gfCNCPoint1[21619] = {X 216.8845, Y 71.0993, Z -2.1667, A 0.000, B 0.000, C 0.000 }
gfCNCPoint1[21620] = {X 215.9082, Y 71.0067, Z -2.1667, A 0.000, B 0.000, C 0.000 }
gfCNCPoint1[21621] = {X 214.2382, Y 70.8314, Z -2.1667, A 0.000, B 0.000, C 0.000 }
gfCNCPoint1[21622] = {X 212.6086, Y 70.4263, Z -2.1667, A 0.000, B 0.000, C 0.000 }
gfCNCPoint1[21623] = {X 211.0509, Y 69.7991, Z -2.1667, A 0.000, B 0.000, C 0.000 }
gfCNCPoint1[21624] = {X 209.5953, Y 68.9620, Z -2.1667, A 0.000, B 0.000, C 0.000 }
gfCNCPoint1[21625] = {X 208.2698, Y 67.9311, Z -2.1667, A 0.000, B 0.000, C 0.000 }
gfCNCPoint1[21626] = {X 207.1000, Y 66.7263, Z -2.1667, A 0.000, B 0.000, C 0.000 }
gfCNCPoint1[21627] = {X 206.1086, Y 65.3710, Z -2.1667, A 0.000, B 0.000, C 0.000 }
gfCNCPoint1[21628] = {X 205.3148, Y 63.8913, Z -2.1667, A 0.000, B 0.000, C 0.000 }
gfCNCPoint1[21629] = {X 204.7338, Y 62.3158, Z -2.1667, A 0.000, B 0.000, C 0.000 }
gfCNCPoint1[21630] = {X 204.3769, Y 60.6750, Z -2.1667, A 0.000, B 0.000, C 0.000 }
gfCNCPoint1[21631] = {X 204.2510, Y 59.0005, Z -2.1667, A 0.000, B 0.000, C 0.000 }
gfCNCPoint1[21632] = {X 204.2508, Y 58.0000, Z -2.1667, A 0.000, B 0.000, C 0.000 }
gfCNCPoint1[21633] = {X 204.3397, Y 56.5375, Z -2.1667, A 0.000, B 0.000, C 0.000 }
gfCNCPoint1[21634] = {X 204.6050, Y 55.0964, Z -2.1667, A 0.000, B 0.000, C 0.000 }
gfCNCPoint1[21635] = {X 205.0427, Y 53.6981, Z -2.1667, A 0.000, B 0.000, C 0.000 }
gfCNCPoint1[21636] = {X 205.6466, Y 52.3631, Z -2.1667, A 0.000, B 0.000, C 0.000 }
gfCNCPoint1[21637] = {X 206.5301, Y 50.9380, Z -2.1667, A 0.000, B 0.000, C 0.000 }
gfCNCPoint1[21638] = {X 207.6024, Y 49.6489, Z -2.1667, A 0.000, B 0.000, C 0.000 }
gfCNCPoint1[21639] = {X 208.8429, Y 48.5207, Z -2.1667, A 0.000, B 0.000, C 0.000 }
gfCNCPoint1[21640] = {X 210.2277, Y 47.5751, Z -2.1667, A 0.000, B 0.000, C 0.000 }
gfCNCPoint1[21641] = {X 209.8801, Y 46.3328, Z -2.1667, A 0.000, B 0.000, C 0.000 }
gfCNCPoint1[21642] = {X 209.7572, Y 45.0487, Z -2.1667, A 0.000, B 0.000, C 0.000 }
gfCNCPoint1[21643] = {X 209.7570, Y 44.1994, Z -2.1667, A 0.000, B 0.000, C 0.000 }
gfCNCPoint1[21644] = {X 209.8559, Y 43.0087, Z -2.1667, A 0.000, B 0.000, C 0.000 }
gfCNCPoint1[21645] = {X 210.1499, Y 41.8506, Z -2.1667, A 0.000, B 0.000, C 0.000 }
gfCNCPoint1[21646] = {X 210.6310, Y 40.7569, Z -2.1667, A 0.000, B 0.000, C 0.000 }
gfCNCPoint1[21647] = {X 211.2859, Y 39.7575, Z -2.1667, A 0.000, B 0.000, C 0.000 }
gfCNCPoint1[21648] = {X 211.2859, Y 37.0789, Z -2.1667, A 0.000, B 0.000, C 0.000 }
gfCNCPoint1[21649] = {X 211.2856, Y 17.4412, Z -2.1667, A 0.000, B 0.000, C 0.000 }
gfCNCPoint1[21650] = {X 210.6368, Y 16.4472, Z -2.1667, A 0.000, B 0.000, C 0.000 }
gfCNCPoint1[21651] = {X 210.1581, Y 15.3610, Z -2.1667, A 0.000, B 0.000, C 0.000 }
gfCNCPoint1[21652] = {X 209.8623, Y 14.2115, Z -2.1667, A 0.000, B 0.000, C 0.000 }
gfCNCPoint1[21653] = {X 209.7572, Y 13.0291, Z -2.1667, A 0.000, B 0.000, C 0.000 }
gfCNCPoint1[21654] = {X 209.7570, Y 12.1868, Z -2.1667, A 0.000, B 0.000, C 0.000 }
gfCNCPoint1[21655] = {X 209.7578, Y 12.0809, Z -2.1667, A 0.000, B 0.000, C 0.000 }
gfCNCPoint1[21656] = {X 209.7601, Y 11.9749, Z -2.1667, A 0.000, B 0.000, C 0.000 }
gfCNCPoint1[21657] = {X 209.9068, Y 10.7178, Z -2.1667, A 0.000, B 0.000, C 0.000 }
gfCNCPoint1[21658] = {X 210.2690, Y 9.5051, Z -2.1667, A 0.000, B 0.000, C 0.000 }
gfCNCPoint1[21659] = {X 207.3611, Y 9.5051, Z -2.1667, A 0.000, B 0.000, C 0.000 }
gfCNCPoint1[21660] = {X 207.3611, Y 7.1051, Z -2.1667, A 0.000, B 0.000, C 0.000 }
gfCNCPoint1[21661] = {X 191.1434, Y 7.1051, Z -2.1667, A 0.000, B 0.000, C 0.000 }
gfCNCPoint1[21662] = {X 193.1003, Y 7.6485, Z -2.1667, A 0.000, B 0.000, C 0.000 }
gfCNCPoint1[21663] = {X 194.9835, Y 8.4087, Z -2.1667, A 0.000, B 0.000, C 0.000 }
gfCNCPoint1[21664] = {X 196.7692, Y 9.3759, Z -2.1667, A 0.000, B 0.000, C 0.000 }
gfCNCPoint1[21665] = {X 198.4348, Y 10.5380, Z -2.1667, A 0.000, B 0.000, C 0.000 }
gfCNCPoint1[21666] = {X 198.8568, Y 10.8884, Z -2.1667, A 0.000, B 0.000, C 0.000 }
gfCNCPoint1[21667] = {X 199.2644, Y 11.2556, Z -2.1667, A 0.000, B 0.000, C 0.000 }
gfCNCPoint1[21668] = {X 200.3494, Y 12.3982, Z -2.1667, A 0.000, B 0.000, C 0.000 }
gfCNCPoint1[21669] = {X 201.2950, Y 13.6586, Z -2.1667, A 0.000, B 0.000, C 0.000 }
gfCNCPoint1[21670] = {X 202.0885, Y 15.0198, Z -2.1667, A 0.000, B 0.000, C 0.000 }
gfCNCPoint1[21671] = {X 202.7195, Y 16.4636, Z -2.1667, A 0.000, B 0.000, C 0.000 }
gfCNCPoint1[21672] = {X 203.2132, Y 18.1834, Z -2.1667, A 0.000, B 0.000, C 0.000 }
gfCNCPoint1[21673] = {X 203.5066, Y 19.9484, Z -2.1667, A 0.000, B 0.000, C 0.000 }
gfCNCPoint1[21674] = {X 203.5957, Y 21.7354, Z -2.1667, A 0.000, B 0.000, C 0.000 }
gfCNCPoint1[21675] = {X 203.4793, Y 23.5208, Z -2.1667, A 0.000, B 0.000, C 0.000 }
gfCNCPoint1[21676] = {X 203.1591, Y 25.2812, Z -2.1667, A 0.000, B 0.000, C 0.000 }
gfCNCPoint1[21677] = {X 202.7588, Y 26.6265, Z -2.1667, A 0.000, B 0.000, C 0.000 }
gfCNCPoint1[21678] = {X 202.2073, Y 27.9172, Z -2.1667, A 0.000, B 0.000, C 0.000 }
gfCNCPoint1[21679] = {X 201.5117, Y 29.1363, Z -2.1667, A 0.000, B 0.000, C 0.000 }
gfCNCPoint1[21680] = {X 200.6812, Y 30.2679, Z -2.1667, A 0.000, B 0.000, C 0.000 }
gfCNCPoint1[21681] = {X 199.7268, Y 31.2971, Z -2.1667, A 0.000, B 0.000, C 0.000 }
gfCNCPoint1[21682] = {X 200.5665, Y 31.8696, Z -2.1667, A 0.000, B 0.000, C 0.000 }
gfCNCPoint1[21683] = {X 201.2694, Y 32.6036, Z -2.1667, A 0.000, B 0.000, C 0.000 }
gfCNCPoint1[21684] = {X 201.8050, Y 33.4674, Z -2.1667, A 0.000, B 0.000, C 0.000 }
gfCNCPoint1[21685] = {X 204.8262, Y 39.7091, Z -2.1667, A 0.000, B 0.000, C 0.000 }
gfCNCPoint1[21686] = {X 205.1508, Y 40.5847, Z -2.1667, A 0.000, B 0.000, C 0.000 }
gfCNCPoint1[21687] = {X 205.3026, Y 41.5062, Z -2.1667, A 0.000, B 0.000, C 0.000 }
gfCNCPoint1[21688] = {X 205.2761, Y 42.4397, Z -2.1667, A 0.000, B 0.000, C 0.000 }
gfCNCPoint1[21689] = {X 205.0723, Y 43.3511, Z -2.1667, A 0.000, B 0.000, C 0.000 }
gfCNCPoint1[21690] = {X 204.6986, Y 44.2070, Z -2.1667, A 0.000, B 0.000, C 0.000 }
gfCNCPoint1[21691] = {X 204.1687, Y 44.9760, Z -2.1667, A 0.000, B 0.000, C 0.000 }
gfCNCPoint1[21692] = {X 203.5020, Y 45.6299, Z -2.1667, A 0.000, B 0.000, C 0.000 }
gfCNCPoint1[21693] = {X 202.9655, Y 46.0637, Z -2.1667, A 0.000, B 0.000, C 0.000 }
gfCNCPoint1[21694] = {X 202.2134, Y 46.5637, Z -2.1667, A 0.000, B 0.000, C 0.000 }
gfCNCPoint1[21695] = {X 201.3821, Y 46.9170, Z -2.1667, A 0.000, B 0.000, C 0.000 }
gfCNCPoint1[21696] = {X 200.5002, Y 47.1116, Z -2.1667, A 0.000, B 0.000, C 0.000 }
gfCNCPoint1[21697] = {X 199.5975, Y 47.1409, Z -2.1667, A 0.000, B 0.000, C 0.000 }
gfCNCPoint1[21698] = {X 198.7048, Y 47.0038, Z -2.1667, A 0.000, B 0.000, C 0.000 }
gfCNCPoint1[21699] = {X 196.3906, Y 48.1788, Z -2.1667, A 0.000, B 0.000, C 0.000 }
gfCNCPoint1[21700] = {X 193.9812, Y 49.1436, Z -2.1667, A 0.000, B 0.000, C 0.000 }
gfCNCPoint1[21701] = {X 191.4956, Y 49.8907, Z -2.1667, A 0.000, B 0.000, C 0.000 }
gfCNCPoint1[21702] = {X 190.2923, Y 50.1563, Z -2.1667, A 0.000, B 0.000, C 0.000 }
gfCNCPoint1[21703] = {X 189.0766, Y 50.3577, Z -2.1667, A 0.000, B 0.000, C 0.000 }
gfCNCPoint1[21704] = {X 186.8979, Y 50.5552, Z -2.1667, A 0.000, B 0.000, C 0.000 }
gfCNCPoint1[21705] = {X 184.7103, Y 50.5468, Z -2.1667, A 0.000, B 0.000, C 0.000 }
gfCNCPoint1[21706] = {X 184.7348, Y 50.0675, Z -2.1667, A 0.000, B 0.000, C 0.000 }
gfCNCPoint1[21707] = {X 183.1149, Y 49.9266, Z -2.1667, A 0.000, B 0.000, C 0.000 }
gfCNCPoint1[21708] = {X 181.5093, Y 49.6703, Z -2.1667, A 0.000, B 0.000, C 0.000 }
gfCNCPoint1[21709] = {X 179.6142, Y 49.1965, Z -2.1667, A 0.000, B 0.000, C 0.000 }
gfCNCPoint1[21710] = {X 177.7853, Y 48.5099, Z -2.1667, A 0.000, B 0.000, C 0.000 }
gfCNCPoint1[21711] = {X 176.0466, Y 47.6193, Z -2.1667, A 0.000, B 0.000, C 0.000 }
gfCNCPoint1[21712] = {X 174.4208, Y 46.5365, Z -2.1667, A 0.000, B 0.000, C 0.000 }
gfCNCPoint1[21713] = {X 173.1808, Y 45.4898, Z -2.1667, A 0.000, B 0.000, C 0.000 }
gfCNCPoint1[21714] = {X 172.0773, Y 44.3002, Z -2.1667, A 0.000, B 0.000, C 0.000 }
gfCNCPoint1[21715] = {X 171.1268, Y 42.9851, Z -2.1667, A 0.000, B 0.000, C 0.000 }
gfCNCPoint1[21716] = {X 170.3432, Y 41.5641, Z -2.1667, A 0.000, B 0.000, C 0.000 }
gfCNCPoint1[21717] = {X 169.7384, Y 40.0584, Z -2.1667, A 0.000, B 0.000, C 0.000 }
gfCNCPoint1[21718] = {X 169.3212, Y 38.4903, Z -2.1667, A 0.000, B 0.000, C 0.000 }
gfCNCPoint1[21719] = {X 169.0979, Y 36.8831, Z -2.1667, A 0.000, B 0.000, C 0.000 }
gfCNCPoint1[21720] = {X 169.0134, Y 35.0395, Z -2.1667, A 0.000, B 0.000, C 0.000 }
gfCNCPoint1[21721] = {X 169.1603, Y 33.2000, Z -2.1667, A 0.000, B 0.000, C 0.000 }
gfCNCPoint1[21722] = {X 169.5364, Y 31.3932, Z -2.1667, A 0.000, B 0.000, C 0.000 }
gfCNCPoint1[21723] = {X 170.1356, Y 29.6478, Z -2.1667, A 0.000, B 0.000, C 0.000 }
gfCNCPoint1[21724] = {X 170.7629, Y 28.3601, Z -2.1667, A 0.000, B 0.000, C 0.000 }
gfCNCPoint1[21725] = {X 171.5529, Y 27.1653, Z -2.1667, A 0.000, B 0.000, C 0.000 }
gfCNCPoint1[21726] = {X 172.4921, Y 26.0840, Z -2.1667, A 0.000, B 0.000, C 0.000 }
gfCNCPoint1[21727] = {X 173.5646, Y 25.1346, Z -2.1667, A 0.000, B 0.000, C 0.000 }
gfCNCPoint1[21728] = {X 174.7519, Y 24.3333, Z -2.1667, A 0.000, B 0.000, C 0.000 }
gfCNCPoint1[21729] = {X 173.9915, Y 23.9230, Z -2.1667, A 0.000, B 0.000, C 0.000 }
gfCNCPoint1[21730] = {X 173.3261, Y 23.3721, Z -2.1667, A 0.000, B 0.000, C 0.000 }
gfCNCPoint1[21731] = {X 172.7811, Y 22.7017, Z -2.1667, A 0.000, B 0.000, C 0.000 }
gfCNCPoint1[21732] = {X 172.3776, Y 21.9378, Z -2.1667, A 0.000, B 0.000, C 0.000 }
gfCNCPoint1[21733] = {X 169.7664, Y 15.5423, Z -2.1667, A 0.000, B 0.000, C 0.000 }
gfCNCPoint1[21734] = {X 169.5126, Y 14.6752, Z -2.1667, A 0.000, B 0.000, C 0.000 }
gfCNCPoint1[21735] = {X 169.4412, Y 13.7745, Z -2.1667, A 0.000, B 0.000, C 0.000 }
gfCNCPoint1[21736] = {X 169.5553, Y 12.8782, Z -2.1667, A 0.000, B 0.000, C 0.000 }
gfCNCPoint1[21737] = {X 169.8501, Y 12.0242, Z -2.1667, A 0.000, B 0.000, C 0.000 }
gfCNCPoint1[21738] = {X 170.3131, Y 11.2483, Z -2.1667, A 0.000, B 0.000, C 0.000 }
gfCNCPoint1[21739] = {X 170.9248, Y 10.5834, Z -2.1667, A 0.000, B 0.000, C 0.000 }
gfCNCPoint1[21740] = {X 171.6594, Y 10.0574, Z -2.1667, A 0.000, B 0.000, C 0.000 }
gfCNCPoint1[21741] = {X 172.2916, Y 9.6970, Z -2.1667, A 0.000, B 0.000, C 0.000 }
gfCNCPoint1[21742] = {X 173.1812, Y 9.3215, Z -2.1667, A 0.000, B 0.000, C 0.000 }
gfCNCPoint1[21743] = {X 174.1312, Y 9.1491, Z -2.1667, A 0.000, B 0.000, C 0.000 }
gfCNCPoint1[21744] = {X 175.0960, Y 9.1881, Z -2.1667, A 0.000, B 0.000, C 0.000 }
gfCNCPoint1[21745] = {X 176.0291, Y 9.4366, Z -2.1667, A 0.000, B 0.000, C 0.000 }
gfCNCPoint1[21746] = {X 178.2250, Y 8.5162, Z -2.1667, A 0.000, B 0.000, C 0.000 }
gfCNCPoint1[21747] = {X 180.5019, Y 7.8195, Z -2.1667, A 0.000, B 0.000, C 0.000 }
gfCNCPoint1[21748] = {X 182.8368, Y 7.3533, Z -2.1667, A 0.000, B 0.000, C 0.000 }
gfCNCPoint1[21749] = {X 185.2066, Y 7.1225, Z -2.1667, A 0.000, B 0.000, C 0.000 }
gfCNCPoint1[21750] = {X 187.5877, Y 7.1291, Z -2.1667, A 0.000, B 0.000, C 0.000 }
gfCNCPoint1[21751] = {X 189.9562, Y 7.3732, Z -2.1667, A 0.000, B 0.000, C 0.000 }
gfCNCPoint1[21752] = {X 191.7220, Y 7.7367, Z -2.1667, A 0.000, B 0.000, C 0.000 }
gfCNCPoint1[21753] = {X 193.4411, Y 8.2794, Z -2.1667, A 0.000, B 0.000, C 0.000 }
gfCNCPoint1[21754] = {X 195.0955, Y 8.9958, Z -2.1667, A 0.000, B 0.000, C 0.000 }
gfCNCPoint1[21755] = {X 196.6676, Y 9.8783, Z -2.1667, A 0.000, B 0.000, C 0.000 }
gfCNCPoint1[21756] = {X 198.1408, Y 10.9175, Z -2.1667, A 0.000, B 0.000, C 0.000 }
gfCNCPoint1[21757] = {X 199.2070, Y 11.8672, Z -2.1667, A 0.000, B 0.000, C 0.000 }
gfCNCPoint1[21758] = {X 200.1638, Y 12.9271, Z -2.1667, A 0.000, B 0.000, C 0.000 }
gfCNCPoint1[21759] = {X 200.9999, Y 14.0847, Z -2.1667, A 0.000, B 0.000, C 0.000 }
gfCNCPoint1[21760] = {X 201.7053, Y 15.3261, Z -2.1667, A 0.000, B 0.000, C 0.000 }
gfCNCPoint1[21761] = {X 202.2717, Y 16.6369, Z -2.1667, A 0.000, B 0.000, C 0.000 }
gfCNCPoint1[21762] = {X 202.7479, Y 18.3014, Z -2.1667, A 0.000, B 0.000, C 0.000 }
gfCNCPoint1[21763] = {X 203.0305, Y 20.0095, Z -2.1667, A 0.000, B 0.000, C 0.000 }
gfCNCPoint1[21764] = {X 203.1157, Y 21.7387, Z -2.1667, A 0.000, B 0.000, C 0.000 }
gfCNCPoint1[21765] = {X 203.0025, Y 23.4663, Z -2.1667, A 0.000, B 0.000, C 0.000 }
gfCNCPoint1[21766] = {X 202.6923, Y 25.1696, Z -2.1667, A 0.000, B 0.000, C 0.000 }
gfCNCPoint1[21767] = {X 202.2576, Y 26.5985, Z -2.1667, A 0.000, B 0.000, C 0.000 }
gfCNCPoint1[21768] = {X 201.6456, Y 27.9610, Z -2.1667, A 0.000, B 0.000, C 0.000 }
gfCNCPoint1[21769] = {X 200.8659, Y 29.2349, Z -2.1667, A 0.000, B 0.000, C 0.000 }
gfCNCPoint1[21770] = {X 199.9311, Y 30.3999, Z -2.1667, A 0.000, B 0.000, C 0.000 }
gfCNCPoint1[21771] = {X 198.8564, Y 31.4371, Z -2.1667, A 0.000, B 0.000, C 0.000 }
gfCNCPoint1[21772] = {X 199.6398, Y 31.7988, Z -2.1667, A 0.000, B 0.000, C 0.000 }
gfCNCPoint1[21773] = {X 200.3375, Y 32.3064, Z -2.1667, A 0.000, B 0.000, C 0.000 }
gfCNCPoint1[21774] = {X 200.9227, Y 32.9404, Z -2.1667, A 0.000, B 0.000, C 0.000 }
gfCNCPoint1[21775] = {X 201.3730, Y 33.6764, Z -2.1667, A 0.000, B 0.000, C 0.000 }
gfCNCPoint1[21776] = {X 204.3942, Y 39.9182, Z -2.1667, A 0.000, B 0.000, C 0.000 }
gfCNCPoint1[21777] = {X 204.7207, Y 40.8441, Z -2.1667, A 0.000, B 0.000, C 0.000 }
gfCNCPoint1[21778] = {X 204.8337, Y 41.8194, Z -2.1667, A 0.000, B 0.000, C 0.000 }
gfCNCPoint1[21779] = {X 204.7276, Y 42.7955, Z -2.1667, A 0.000, B 0.000, C 0.000 }
gfCNCPoint1[21780] = {X 204.4078, Y 43.7238, Z -2.1667, A 0.000, B 0.000, C 0.000 }
gfCNCPoint1[21781] = {X 203.8900, Y 44.5580, Z -2.1667, A 0.000, B 0.000, C 0.000 }
gfCNCPoint1[21782] = {X 203.2002, Y 45.2567, Z -2.1667, A 0.000, B 0.000, C 0.000 }
gfCNCPoint1[21783] = {X 202.6637, Y 45.6904, Z -2.1667, A 0.000, B 0.000, C 0.000 }
gfCNCPoint1[21784] = {X 201.9521, Y 46.1590, Z -2.1667, A 0.000, B 0.000, C 0.000 }
gfCNCPoint1[21785] = {X 201.1638, Y 46.4822, Z -2.1667, A 0.000, B 0.000, C 0.000 }
gfCNCPoint1[21786] = {X 200.3280, Y 46.6480, Z -2.1667, A 0.000, B 0.000, C 0.000 }
gfCNCPoint1[21787] = {X 199.4760, Y 46.6501, Z -2.1667, A 0.000, B 0.000, C 0.000 }
gfCNCPoint1[21788] = {X 198.6394, Y 46.4887, Z -2.1667, A 0.000, B 0.000, C 0.000 }
gfCNCPoint1[21789] = {X 196.3113, Y 47.6875, Z -2.1667, A 0.000, B 0.000, C 0.000 }
gfCNCPoint1[21790] = {X 193.8835, Y 48.6692, Z -2.1667, A 0.000, B 0.000, C 0.000 }
gfCNCPoint1[21791] = {X 191.3765, Y 49.4257, Z -2.1667, A 0.000, B 0.000, C 0.000 }
gfCNCPoint1[21792] = {X 189.1872, Y 49.8571, Z -2.1667, A 0.000, B 0.000, C 0.000 }
gfCNCPoint1[21793] = {X 186.9662, Y 50.0717, Z -2.1667, A 0.000, B 0.000, C 0.000 }
gfCNCPoint1[21794] = {X 184.7348, Y 50.0675, Z -2.1667, A 0.000, B 0.000, C 0.000 }
gfCNCPoint1[21795] = {X 184.7103, Y 50.5468, Z -2.1667, A 0.000, B 0.000, C 0.000 }
gfCNCPoint1[21796] = {X 185.7068, Y 51.5003, Z -2.1667, A 0.000, B 0.000, C 0.000 }
gfCNCPoint1[21797] = {X 186.5577, Y 52.5857, Z -2.1667, A 0.000, B 0.000, C 0.000 }
gfCNCPoint1[21798] = {X 187.2457, Y 53.7810, Z -2.1667, A 0.000, B 0.000, C 0.000 }
gfCNCPoint1[21799] = {X 187.7793, Y 55.1333, Z -2.1667, A 0.000, B 0.000, C 0.000 }
gfCNCPoint1[21800] = {X 188.1043, Y 56.5503, Z -2.1667, A 0.000, B 0.000, C 0.000 }
gfCNCPoint1[21801] = {X 188.2135, Y 58.0000, Z -2.1667, A 0.000, B 0.000, C 0.000 }
gfCNCPoint1[21802] = {X 188.2132, Y 59.0140, Z -2.1667, A 0.000, B 0.000, C 0.000 }
gfCNCPoint1[21803] = {X 188.2026, Y 59.3931, Z -2.1667, A 0.000, B 0.000, C 0.000 }
gfCNCPoint1[21804] = {X 188.1772, Y 59.7715, Z -2.1667, A 0.000, B 0.000, C 0.000 }
gfCNCPoint1[21805] = {X 213.5228, Y 87.4328, Z -2.1667, A 0.000, B 0.000, C 0.000 }
gfCNCPoint1[21806] = {X 214.2178, Y 87.3803, Z -2.1667, A 0.000, B 0.000, C 0.000 }
gfCNCPoint1[21807] = {X 214.9136, Y 87.3388, Z -2.1667, A 0.000, B 0.000, C 0.000 }
gfCNCPoint1[21808] = {X 234.0929, Y 75.0516, Z -2.1667, A 0.000, B 0.000, C 0.000 }
gfCNCPoint1[21809] = {X 219.6587, Y 69.3868, Z -2.1667, A 0.000, B 0.000, C 0.000 }
gfCNCPoint1[21810] = {X 218.4698, Y 68.9869, Z -2.1667, A 0.000, B 0.000, C 0.000 }
gfCNCPoint1[21811] = {X 217.2429, Y 68.7262, Z -2.1667, A 0.000, B 0.000, C 0.000 }
gfCNCPoint1[21812] = {X 215.9942, Y 68.6082, Z -2.1667, A 0.000, B 0.000, C 0.000 }
gfCNCPoint1[21813] = {X 214.5238, Y 68.4439, Z -2.1667, A 0.000, B 0.000, C 0.000 }
gfCNCPoint1[21814] = {X 213.0956, Y 68.0575, Z -2.1667, A 0.000, B 0.000, C 0.000 }
gfCNCPoint1[21815] = {X 211.7431, Y 67.4579, Z -2.1667, A 0.000, B 0.000, C 0.000 }
gfCNCPoint1[21816] = {X 210.4977, Y 66.6591, Z -2.1667, A 0.000, B 0.000, C 0.000 }
gfCNCPoint1[21817] = {X 209.3885, Y 65.6800, Z -2.1667, A 0.000, B 0.000, C 0.000 }
gfCNCPoint1[21818] = {X 208.4416, Y 64.5432, Z -2.1667, A 0.000, B 0.000, C 0.000 }
gfCNCPoint1[21819] = {X 207.6789, Y 63.2754, Z -2.1667, A 0.000, B 0.000, C 0.000 }
gfCNCPoint1[21820] = {X 207.1184, Y 61.9061, Z -2.1667, A 0.000, B 0.000, C 0.000 }
gfCNCPoint1[21821] = {X 206.7730, Y 60.4675, Z -2.1667, A 0.000, B 0.000, C 0.000 }
gfCNCPoint1[21822] = {X 206.6510, Y 58.9930, Z -2.1667, A 0.000, B 0.000, C 0.000 }
gfCNCPoint1[21823] = {X 206.6508, Y 58.0000, Z -2.1667, A 0.000, B 0.000, C 0.000 }
gfCNCPoint1[21824] = {X 206.7577, Y 56.5655, Z -2.1667, A 0.000, B 0.000, C 0.000 }
gfCNCPoint1[21825] = {X 207.0759, Y 55.1628, Z -2.1667, A 0.000, B 0.000, C 0.000 }
gfCNCPoint1[21826] = {X 207.5986, Y 53.8226, Z -2.1667, A 0.000, B 0.000, C 0.000 }
gfCNCPoint1[21827] = {X 208.3140, Y 52.5747, Z -2.1667, A 0.000, B 0.000, C 0.000 }
gfCNCPoint1[21828] = {X 209.2065, Y 51.4466, Z -2.1667, A 0.000, B 0.000, C 0.000 }
gfCNCPoint1[21829] = {X 210.2563, Y 50.4632, Z -2.1667, A 0.000, B 0.000, C 0.000 }
gfCNCPoint1[21830] = {X 211.4402, Y 49.6463, Z -2.1667, A 0.000, B 0.000, C 0.000 }
gfCNCPoint1[21831] = {X 212.5893, Y 49.0723, Z -2.1667, A 0.000, B 0.000, C 0.000 }
gfCNCPoint1[21832] = {X 213.8042, Y 48.6556, Z -2.1667, A 0.000, B 0.000, C 0.000 }
gfCNCPoint1[21833] = {X 213.2578, Y 48.0874, Z -2.1667, A 0.000, B 0.000, C 0.000 }
gfCNCPoint1[21834] = {X 212.8100, Y 47.4386, Z -2.1667, A 0.000, B 0.000, C 0.000 }
gfCNCPoint1[21835] = {X 212.4725, Y 46.7262, Z -2.1667, A 0.000, B 0.000, C 0.000 }
gfCNCPoint1[21836] = {X 212.2401, Y 45.8965, Z -2.1667, A 0.000, B 0.000, C 0.000 }
gfCNCPoint1[21837] = {X 212.1572, Y 45.0389, Z -2.1667, A 0.000, B 0.000, C 0.000 }
gfCNCPoint1[21838] = {X 212.1570, Y 44.1994, Z -2.1667, A 0.000, B 0.000, C 0.000 }
gfCNCPoint1[21839] = {X 212.2384, Y 43.3175, Z -2.1667, A 0.000, B 0.000, C 0.000 }
gfCNCPoint1[21840] = {X 212.4799, Y 42.4654, Z -2.1667, A 0.000, B 0.000, C 0.000 }
gfCNCPoint1[21841] = {X 212.8733, Y 41.6720, Z -2.1667, A 0.000, B 0.000, C 0.000 }
gfCNCPoint1[21842] = {X 213.4053, Y 40.9639, Z -2.1667, A 0.000, B 0.000, C 0.000 }
gfCNCPoint1[21843] = {X 213.6831, Y 40.6575, Z -2.1667, A 0.000, B 0.000, C 0.000 }
gfCNCPoint1[21844] = {X 213.6859, Y 40.3041, Z -2.1667, A 0.000, B 0.000, C 0.000 }
gfCNCPoint1[21845] = {X 213.6859, Y 17.4645, Z -2.1667, A 0.000, B 0.000, C 0.000 }
gfCNCPoint1[21846] = {X 213.6805, Y 16.7698, Z -2.1667, A 0.000, B 0.000, C 0.000 }
gfCNCPoint1[21847] = {X 213.6802, Y 16.5201, Z -2.1667, A 0.000, B 0.000, C 0.000 }
gfCNCPoint1[21848] = {X 213.0407, Y 15.7787, Z -2.1667, A 0.000, B 0.000, C 0.000 }
gfCNCPoint1[21849] = {X 212.5621, Y 14.9246, Z -2.1667, A 0.000, B 0.000, C 0.000 }
gfCNCPoint1[21850] = {X 212.2635, Y 13.9921, Z -2.1667, A 0.000, B 0.000, C 0.000 }
gfCNCPoint1[21851] = {X 212.1572, Y 13.0188, Z -2.1667, A 0.000, B 0.000, C 0.000 }
gfCNCPoint1[21852] = {X 212.1570, Y 12.1868, Z -2.1667, A 0.000, B 0.000, C 0.000 }
gfCNCPoint1[21853] = {X 212.2436, Y 11.2718, Z -2.1667, A 0.000, B 0.000, C 0.000 }
gfCNCPoint1[21854] = {X 212.5002, Y 10.3892, Z -2.1667, A 0.000, B 0.000, C 0.000 }
gfCNCPoint1[21855] = {X 212.9449, Y 9.5281, Z -2.1667, A 0.000, B 0.000, C 0.000 }
gfCNCPoint1[21856] = {X 213.5510, Y 8.7718, Z -2.1667, A 0.000, B 0.000, C 0.000 }
gfCNCPoint1[21857] = {X 214.2946, Y 8.1503, Z -2.1667, A 0.000, B 0.000, C 0.000 }
gfCNCPoint1[21858] = {X 215.1463, Y 7.6880, Z -2.1667, A 0.000, B 0.000, C 0.000 }
gfCNCPoint1[21859] = {X 216.0727, Y 7.4030, Z -2.1667, A 0.000, B 0.000, C 0.000 }
gfCNCPoint1[21860] = {X 217.0370, Y 7.3068, Z -2.1667, A 0.000, B 0.000, C 0.000 }
gfCNCPoint1[21861] = {X 223.4805, Y 7.3068, Z -2.1667, A 0.000, B 0.000, C 0.000 }
gfCNCPoint1[21862] = {X 224.4448, Y 7.4030, Z -2.1667, A 0.000, B 0.000, C 0.000 }
gfCNCPoint1[21863] = {X 225.3712, Y 7.6880, Z -2.1667, A 0.000, B 0.000, C 0.000 }
gfCNCPoint1[21864] = {X 226.2229, Y 8.1503, Z -2.1667, A 0.000, B 0.000, C 0.000 }
gfCNCPoint1[21865] = {X 226.9665, Y 8.7718, Z -2.1667, A 0.000, B 0.000, C 0.000 }
gfCNCPoint1[21866] = {X 227.5726, Y 9.5281, Z -2.1667, A 0.000, B 0.000, C 0.000 }
gfCNCPoint1[21867] = {X 228.0173, Y 10.3892, Z -2.1667, A 0.000, B 0.000, C 0.000 }
gfCNCPoint1[21868] = {X 228.2739, Y 11.2718, Z -2.1667, A 0.000, B 0.000, C 0.000 }
gfCNCPoint1[21869] = {X 228.3605, Y 12.1868, Z -2.1667, A 0.000, B 0.000, C 0.000 }
gfCNCPoint1[21870] = {X 228.3603, Y 13.0237, Z -2.1667, A 0.000, B 0.000, C 0.000 }
gfCNCPoint1[21871] = {X 228.2528, Y 13.9974, Z -2.1667, A 0.000, B 0.000, C 0.000 }
gfCNCPoint1[21872] = {X 227.9531, Y 14.9300, Z -2.1667, A 0.000, B 0.000, C 0.000 }
gfCNCPoint1[21873] = {X 227.4732, Y 15.7839, Z -2.1667, A 0.000, B 0.000, C 0.000 }
gfCNCPoint1[21874] = {X 226.8323, Y 16.5248, Z -2.1667, A 0.000, B 0.000, C 0.000 }
gfCNCPoint1[21875] = {X 226.8332, Y 40.6629, Z -2.1667, A 0.000, B 0.000, C 0.000 }
gfCNCPoint1[21876] = {X 227.4738, Y 41.4038, Z -2.1667, A 0.000, B 0.000, C 0.000 }
gfCNCPoint1[21877] = {X 227.9535, Y 42.2577, Z -2.1667, A 0.000, B 0.000, C 0.000 }
gfCNCPoint1[21878] = {X 228.2530, Y 43.1903, Z -2.1667, A 0.000, B 0.000, C 0.000 }
gfCNCPoint1[21879] = {X 228.3603, Y 44.1638, Z -2.1667, A 0.000, B 0.000, C 0.000 }
gfCNCPoint1[21880] = {X 228.3605, Y 45.0000, Z -2.1667, A 0.000, B 0.000, C 0.000 }
gfCNCPoint1[21881] = {X 228.3507, Y 45.3090, Z -2.1667, A 0.000, B 0.000, C 0.000 }
gfCNCPoint1[21882] = {X 228.3214, Y 45.6167, Z -2.1667, A 0.000, B 0.000, C 0.000 }
gfCNCPoint1[21883] = {X 228.0910, Y 46.5992, Z -2.1667, A 0.000, B 0.000, C 0.000 }
gfCNCPoint1[21884] = {X 227.6635, Y 47.5134, Z -2.1667, A 0.000, B 0.000, C 0.000 }
gfCNCPoint1[21885] = {X 227.0571, Y 48.3200, Z -2.1667, A 0.000, B 0.000, C 0.000 }
gfCNCPoint1[21886] = {X 226.7053, Y 47.9934, Z -2.1667, A 0.000, B 0.000, C 0.000 }
gfCNCPoint1[21887] = {X 226.0261, Y 48.5889, Z -2.1667, A 0.000, B 0.000, C 0.000 }
gfCNCPoint1[21888] = {X 225.2396, Y 49.0331, Z -2.1667, A 0.000, B 0.000, C 0.000 }
gfCNCPoint1[21889] = {X 224.3790, Y 49.3073, Z -2.1667, A 0.000, B 0.000, C 0.000 }
gfCNCPoint1[21890] = {X 223.4805, Y 49.4000, Z -2.1667, A 0.000, B 0.000, C 0.000 }
gfCNCPoint1[21891] = {X 217.0370, Y 49.4000, Z -2.1667, A 0.000, B 0.000, C 0.000 }
gfCNCPoint1[21892] = {X 216.0579, Y 49.2897, Z -2.1667, A 0.000, B 0.000, C 0.000 }
gfCNCPoint1[21893] = {X 215.1279, Y 48.9643, Z -2.1667, A 0.000, B 0.000, C 0.000 }
gfCNCPoint1[21894] = {X 214.2936, Y 48.4400, Z -2.1667, A 0.000, B 0.000, C 0.000 }
gfCNCPoint1[21895] = {X 213.5969, Y 47.7433, Z -2.1667, A 0.000, B 0.000, C 0.000 }
gfCNCPoint1[21896] = {X 213.0727, Y 46.9091, Z -2.1667, A 0.000, B 0.000, C 0.000 }
gfCNCPoint1[21897] = {X 212.7473, Y 45.9791, Z -2.1667, A 0.000, B 0.000, C 0.000 }
gfCNCPoint1[21898] = {X 212.6370, Y 45.0000, Z -2.1667, A 0.000, B 0.000, C 0.000 }
gfCNCPoint1[21899] = {X 212.6370, Y 44.1994, Z -2.1667, A 0.000, B 0.000, C 0.000 }
gfCNCPoint1[21900] = {X 212.7103, Y 43.4054, Z -2.1667, A 0.000, B 0.000, C 0.000 }
gfCNCPoint1[21901] = {X 212.9277, Y 42.6382, Z -2.1667, A 0.000, B 0.000, C 0.000 }
gfCNCPoint1[21902] = {X 213.2819, Y 41.9238, Z -2.1667, A 0.000, B 0.000, C 0.000 }
gfCNCPoint1[21903] = {X 213.7609, Y 41.2863, Z -2.1667, A 0.000, B 0.000, C 0.000 }
gfCNCPoint1[21904] = {X 214.1617, Y 40.8442, Z -2.1667, A 0.000, B 0.000, C 0.000 }
gfCNCPoint1[21905] = {X 214.1659, Y 40.3060, Z -2.1667, A 0.000, B 0.000, C 0.000 }
gfCNCPoint1[21906] = {X 214.1659, Y 17.4626, Z -2.1667, A 0.000, B 0.000, C 0.000 }
gfCNCPoint1[21907] = {X 214.1605, Y 16.7692, Z -2.1667, A 0.000, B 0.000, C 0.000 }
gfCNCPoint1[21908] = {X 214.1600, Y 16.3071, Z -2.1667, A 0.000, B 0.000, C 0.000 }
gfCNCPoint1[21909] = {X 213.5172, Y 15.6183, Z -2.1667, A 0.000, B 0.000, C 0.000 }
gfCNCPoint1[21910] = {X 213.0358, Y 14.8084, Z -2.1667, A 0.000, B 0.000, C 0.000 }
gfCNCPoint1[21911] = {X 212.7379, Y 13.9146, Z -2.1667, A 0.000, B 0.000, C 0.000 }
gfCNCPoint1[21912] = {X 212.6370, Y 12.9779, Z -2.1667, A 0.000, B 0.000, C 0.000 }
gfCNCPoint1[21913] = {X 212.6370, Y 12.1868, Z -2.1667, A 0.000, B 0.000, C 0.000 }
gfCNCPoint1[21914] = {X 212.7473, Y 11.2077, Z -2.1667, A 0.000, B 0.000, C 0.000 }
gfCNCPoint1[21915] = {X 213.0728, Y 10.2777, Z -2.1667, A 0.000, B 0.000, C 0.000 }
gfCNCPoint1[21916] = {X 213.5970, Y 9.4435, Z -2.1667, A 0.000, B 0.000, C 0.000 }
gfCNCPoint1[21917] = {X 214.2937, Y 8.7468, Z -2.1667, A 0.000, B 0.000, C 0.000 }
gfCNCPoint1[21918] = {X 215.1279, Y 8.2226, Z -2.1667, A 0.000, B 0.000, C 0.000 }
gfCNCPoint1[21919] = {X 216.0579, Y 7.8971, Z -2.1667, A 0.000, B 0.000, C 0.000 }
gfCNCPoint1[21920] = {X 217.0370, Y 7.7868, Z -2.1667, A 0.000, B 0.000, C 0.000 }
gfCNCPoint1[21921] = {X 223.4805, Y 7.7868, Z -2.1667, A 0.000, B 0.000, C 0.000 }
gfCNCPoint1[21922] = {X 224.4596, Y 7.8971, Z -2.1667, A 0.000, B 0.000, C 0.000 }
gfCNCPoint1[21923] = {X 225.3896, Y 8.2226, Z -2.1667, A 0.000, B 0.000, C 0.000 }
gfCNCPoint1[21924] = {X 226.2238, Y 8.7468, Z -2.1667, A 0.000, B 0.000, C 0.000 }
gfCNCPoint1[21925] = {X 226.9205, Y 9.4435, Z -2.1667, A 0.000, B 0.000, C 0.000 }
gfCNCPoint1[21926] = {X 227.4447, Y 10.2777, Z -2.1667, A 0.000, B 0.000, C 0.000 }
gfCNCPoint1[21927] = {X 227.7702, Y 11.2077, Z -2.1667, A 0.000, B 0.000, C 0.000 }
gfCNCPoint1[21928] = {X 227.8805, Y 12.1868, Z -2.1667, A 0.000, B 0.000, C 0.000 }
gfCNCPoint1[21929] = {X 227.8802, Y 13.0233, Z -2.1667, A 0.000, B 0.000, C 0.000 }
gfCNCPoint1[21930] = {X 227.7719, Y 13.9495, Z -2.1667, A 0.000, B 0.000, C 0.000 }
gfCNCPoint1[21931] = {X 227.4708, Y 14.8321, Z -2.1667, A 0.000, B 0.000, C 0.000 }
gfCNCPoint1[21932] = {X 226.9904, Y 15.6314, Z -2.1667, A 0.000, B 0.000, C 0.000 }
gfCNCPoint1[21933] = {X 226.3523, Y 16.3116, Z -2.1667, A 0.000, B 0.000, C 0.000 }
gfCNCPoint1[21934] = {X 226.3532, Y 40.8760, Z -2.1667, A 0.000, B 0.000, C 0.000 }
gfCNCPoint1[21935] = {X 226.9978, Y 41.5652, Z -2.1667, A 0.000, B 0.000, C 0.000 }
gfCNCPoint1[21936] = {X 227.4805, Y 42.3758, Z -2.1667, A 0.000, B 0.000, C 0.000 }
gfCNCPoint1[21937] = {X 227.7793, Y 43.2708, Z -2.1667, A 0.000, B 0.000, C 0.000 }
gfCNCPoint1[21938] = {X 227.8805, Y 44.2089, Z -2.1667, A 0.000, B 0.000, C 0.000 }
gfCNCPoint1[21939] = {X 227.8805, Y 45.0000, Z -2.1667, A 0.000, B 0.000, C 0.000 }
gfCNCPoint1[21940] = {X 227.8037, Y 45.8182, Z -2.1667, A 0.000, B 0.000, C 0.000 }
gfCNCPoint1[21941] = {X 227.5762, Y 46.6079, Z -2.1667, A 0.000, B 0.000, C 0.000 }
gfCNCPoint1[21942] = {X 227.2057, Y 47.3415, Z -2.1667, A 0.000, B 0.000, C 0.000 }
gfCNCPoint1[21943] = {X 226.7053, Y 47.9934, Z -2.1667, A 0.000, B 0.000, C 0.000 }
gfCNCPoint1[21944] = {X 227.0571, Y 48.3200, Z -2.1667, A 0.000, B 0.000, C 0.000 }
gfCNCPoint1[21945] = {X 236.2309, Y 48.3200, Z -2.1667, A 0.000, B 0.000, C 0.000 }
gfCNCPoint1[21946] = {X 235.6245, Y 47.5134, Z -2.1667, A 0.000, B 0.000, C 0.000 }
gfCNCPoint1[21947] = {X 235.1970, Y 46.5992, Z -2.1667, A 0.000, B 0.000, C 0.000 }
gfCNCPoint1[21948] = {X 234.9666, Y 45.6167, Z -2.1667, A 0.000, B 0.000, C 0.000 }
gfCNCPoint1[21949] = {X 234.9373, Y 45.3090, Z -2.1667, A 0.000, B 0.000, C 0.000 }
gfCNCPoint1[21950] = {X 234.9275, Y 45.0000, Z -2.1667, A 0.000, B 0.000, C 0.000 }
gfCNCPoint1[21951] = {X 234.9275, Y 44.2089, Z -2.1667, A 0.000, B 0.000, C 0.000 }
gfCNCPoint1[21952] = {X 235.0194, Y 43.2661, Z -2.1667, A 0.000, B 0.000, C 0.000 }
gfCNCPoint1[21953] = {X 235.2917, Y 42.3588, Z -2.1667, A 0.000, B 0.000, C 0.000 }
gfCNCPoint1[21954] = {X 235.7342, Y 41.5213, Z -2.1667, A 0.000, B 0.000, C 0.000 }
gfCNCPoint1[21955] = {X 236.3302, Y 40.7849, Z -2.1667, A 0.000, B 0.000, C 0.000 }
gfCNCPoint1[21956] = {X 237.0572, Y 40.1776, Z -2.1667, A 0.000, B 0.000, C 0.000 }
gfCNCPoint1[21957] = {X 237.8878, Y 39.7222, Z -2.1667, A 0.000, B 0.000, C 0.000 }
gfCNCPoint1[21958] = {X 241.5467, Y 32.5603, Z -2.1667, A 0.000, B 0.000, C 0.000 }
gfCNCPoint1[21959] = {X 240.2124, Y 31.5577, Z -2.1667, A 0.000, B 0.000, C 0.000 }
gfCNCPoint1[21960] = {X 239.0318, Y 30.3779, Z -2.1667, A 0.000, B 0.000, C 0.000 }
gfCNCPoint1[21961] = {X 238.0282, Y 29.0444, Z -2.1667, A 0.000, B 0.000, C 0.000 }
gfCNCPoint1[21962] = {X 237.2215, Y 27.5832, Z -2.1667, A 0.000, B 0.000, C 0.000 }
gfCNCPoint1[21963] = {X 236.6275, Y 26.0235, Z -2.1667, A 0.000, B 0.000, C 0.000 }
gfCNCPoint1[21964] = {X 236.1924, Y 24.1499, Z -2.1667, A 0.000, B 0.000, C 0.000 }
gfCNCPoint1[21965] = {X 235.9705, Y 22.2393, Z -2.1667, A 0.000, B 0.000, C 0.000 }
gfCNCPoint1[21966] = {X 235.9646, Y 20.3158, Z -2.1667, A 0.000, B 0.000, C 0.000 }
gfCNCPoint1[21967] = {X 236.1749, Y 18.4039, Z -2.1667, A 0.000, B 0.000, C 0.000 }
gfCNCPoint1[21968] = {X 236.5985, Y 16.5277, Z -2.1667, A 0.000, B 0.000, C 0.000 }
gfCNCPoint1[21969] = {X 237.1178, Y 15.0571, Z -2.1667, A 0.000, B 0.000, C 0.000 }
gfCNCPoint1[21970] = {X 237.8175, Y 13.6633, Z -2.1667, A 0.000, B 0.000, C 0.000 }
gfCNCPoint1[21971] = {X 238.6865, Y 12.3682, Z -2.1667, A 0.000, B 0.000, C 0.000 }
gfCNCPoint1[21972] = {X 239.7111, Y 11.1925, Z -2.1667, A 0.000, B 0.000, C 0.000 }
gfCNCPoint1[21973] = {X 240.8753, Y 10.1545, Z -2.1667, A 0.000, B 0.000, C 0.000 }
gfCNCPoint1[21974] = {X 242.1604, Y 9.2707, Z -2.1667, A 0.000, B 0.000, C 0.000 }
gfCNCPoint1[21975] = {X 243.5464, Y 8.5553, Z -2.1667, A 0.000, B 0.000, C 0.000 }
gfCNCPoint1[21976] = {X 245.0111, Y 8.0194, Z -2.1667, A 0.000, B 0.000, C 0.000 }
gfCNCPoint1[21977] = {X 246.5315, Y 7.6715, Z -2.1667, A 0.000, B 0.000, C 0.000 }
gfCNCPoint1[21978] = {X 248.6761, Y 7.3937, Z -2.1667, A 0.000, B 0.000, C 0.000 }
gfCNCPoint1[21979] = {X 250.8370, Y 7.3116, Z -2.1667, A 0.000, B 0.000, C 0.000 }
gfCNCPoint1[21980] = {X 266.7608, Y 7.3116, Z -2.1667, A 0.000, B 0.000, C 0.000 }
gfCNCPoint1[21981] = {X 267.7190, Y 7.4130, Z -2.1667, A 0.000, B 0.000, C 0.000 }
gfCNCPoint1[21982] = {X 268.6386, Y 7.7006, Z -2.1667, A 0.000, B 0.000, C 0.000 }
gfCNCPoint1[21983] = {X 269.4838, Y 8.1632, Z -2.1667, A 0.000, B 0.000, C 0.000 }
gfCNCPoint1[21984] = {X 270.2217, Y 8.7828, Z -2.1667, A 0.000, B 0.000, C 0.000 }
gfCNCPoint1[21985] = {X 270.8236, Y 9.5353, Z -2.1667, A 0.000, B 0.000, C 0.000 }
gfCNCPoint1[21986] = {X 271.2660, Y 10.3913, Z -2.1667, A 0.000, B 0.000, C 0.000 }
gfCNCPoint1[21987] = {X 271.5232, Y 11.2720, Z -2.1667, A 0.000, B 0.000, C 0.000 }
gfCNCPoint1[21988] = {X 271.6110, Y 12.1853, Z -2.1667, A 0.000, B 0.000, C 0.000 }
gfCNCPoint1[21989] = {X 271.6108, Y 13.0282, Z -2.1667, A 0.000, B 0.000, C 0.000 }
gfCNCPoint1[21990] = {X 271.5123, Y 13.9546, Z -2.1667, A 0.000, B 0.000, C 0.000 }
gfCNCPoint1[21991] = {X 271.2396, Y 14.8453, Z -2.1667, A 0.000, B 0.000, C 0.000 }
gfCNCPoint1[21992] = {X 275.6743, Y 16.6820, Z -2.1667, A 0.000, B 0.000, C 0.000 }
gfCNCPoint1[21993] = {X 275.3123, Y 17.4574, Z -2.1667, A 0.000, B 0.000, C 0.000 }
gfCNCPoint1[21994] = {X 274.8831, Y 18.1978, Z -2.1667, A 0.000, B 0.000, C 0.000 }
gfCNCPoint1[21995] = {X 274.8830, Y 38.9888, Z -2.1667, A 0.000, B 0.000, C 0.000 }
gfCNCPoint1[21996] = {X 275.3139, Y 39.7325, Z -2.1667, A 0.000, B 0.000, C 0.000 }
gfCNCPoint1[21997] = {X 275.6771, Y 40.5115, Z -2.1667, A 0.000, B 0.000, C 0.000 }
gfCNCPoint1[21998] = {X 276.0384, Y 39.7367, Z -2.1667, A 0.000, B 0.000, C 0.000 }
gfCNCPoint1[21999] = {X 276.4662, Y 38.9965, Z -2.1667, A 0.000, B 0.000, C 0.000 }
gfCNCPoint1[22000] = {X 276.4658, Y 18.1982, Z -2.1667, A 0.000, B 0.000, C 0.000 }
gfCNCPoint1[22001] = {X 276.0365, Y 17.4576, Z -2.1667, A 0.000, B 0.000, C 0.000 }
gfCNCPoint1[22002] = {X 275.6743, Y 16.6820, Z -2.1667, A 0.000, B 0.000, C 0.000 }
gfCNCPoint1[22003] = {X 273.4570, Y 15.7637, Z -2.1667, A 0.000, B 0.000, C 0.000 }
gfCNCPoint1[22004] = {X 273.0261, Y 16.6345, Z -2.1667, A 0.000, B 0.000, C 0.000 }
gfCNCPoint1[22005] = {X 272.4831, Y 17.4403, Z -2.1667, A 0.000, B 0.000, C 0.000 }
gfCNCPoint1[22006] = {X 272.4830, Y 39.7463, Z -2.1667, A 0.000, B 0.000, C 0.000 }
gfCNCPoint1[22007] = {X 273.0274, Y 40.5545, Z -2.1667, A 0.000, B 0.000, C 0.000 }
gfCNCPoint1[22008] = {X 273.4591, Y 41.4282, Z -2.1667, A 0.000, B 0.000, C 0.000 }
gfCNCPoint1[22009] = {X 273.7590, Y 42.3100, Z -2.1667, A 0.000, B 0.000, C 0.000 }
gfCNCPoint1[22010] = {X 273.9440, Y 43.2228, Z -2.1667, A 0.000, B 0.000, C 0.000 }
gfCNCPoint1[22011] = {X 274.0108, Y 44.1519, Z -2.1667, A 0.000, B 0.000, C 0.000 }
gfCNCPoint1[22012] = {X 274.0110, Y 45.0000, Z -2.1667, A 0.000, B 0.000, C 0.000 }
gfCNCPoint1[22013] = {X 273.9884, Y 45.5734, Z -2.1667, A 0.000, B 0.000, C 0.000 }
gfCNCPoint1[22014] = {X 273.9207, Y 46.1433, Z -2.1667, A 0.000, B 0.000, C 0.000 }
gfCNCPoint1[22015] = {X 275.0713, Y 45.9760, Z -2.1667, A 0.000, B 0.000, C 0.000 }
gfCNCPoint1[22016] = {X 276.2327, Y 45.9200, Z -2.1667, A 0.000, B 0.000, C 0.000 }
gfCNCPoint1[22017] = {X 277.3960, Y 45.9200, Z -2.1667, A 0.000, B 0.000, C 0.000 }
gfCNCPoint1[22018] = {X 277.3539, Y 45.4857, Z -2.1667, A 0.000, B 0.000, C 0.000 }
gfCNCPoint1[22019] = {X 277.3378, Y 45.0497, Z -2.1667, A 0.000, B 0.000, C 0.000 }
gfCNCPoint1[22020] = {X 277.3377, Y 44.1969, Z -2.1667, A 0.000, B 0.000, C 0.000 }
gfCNCPoint1[22021] = {X 277.4034, Y 43.2528, Z -2.1667, A 0.000, B 0.000, C 0.000 }
gfCNCPoint1[22022] = {X 277.5901, Y 42.3251, Z -2.1667, A 0.000, B 0.000, C 0.000 }
gfCNCPoint1[22023] = {X 277.8948, Y 41.4291, Z -2.1667, A 0.000, B 0.000, C 0.000 }
gfCNCPoint1[22024] = {X 278.3248, Y 40.5581, Z -2.1667, A 0.000, B 0.000, C 0.000 }
gfCNCPoint1[22025] = {X 278.8662, Y 39.7516, Z -2.1667, A 0.000, B 0.000, C 0.000 }
gfCNCPoint1[22026] = {X 278.8658, Y 17.4406, Z -2.1667, A 0.000, B 0.000, C 0.000 }
gfCNCPoint1[22027] = {X 278.3227, Y 16.6347, Z -2.1667, A 0.000, B 0.000, C 0.000 }
gfCNCPoint1[22028] = {X 277.8917, Y 15.7637, Z -2.1667, A 0.000, B 0.000, C 0.000 }
gfCNCPoint1[22029] = {X 277.5902, Y 14.8788, Z -2.1667, A 0.000, B 0.000, C 0.000 }
gfCNCPoint1[22030] = {X 277.4046, Y 13.9627, Z -2.1667, A 0.000, B 0.000, C 0.000 }
gfCNCPoint1[22031] = {X 277.3379, Y 13.0303, Z -2.1667, A 0.000, B 0.000, C 0.000 }
gfCNCPoint1[22032] = {X 277.3377, Y 12.1868, Z -2.1667, A 0.000, B 0.000, C 0.000 }
gfCNCPoint1[22033] = {X 277.3952, Y 11.2737, Z -2.1667, A 0.000, B 0.000, C 0.000 }
gfCNCPoint1[22034] = {X 277.5667, Y 10.3751, Z -2.1667, A 0.000, B 0.000, C 0.000 }
gfCNCPoint1[22035] = {X 277.8496, Y 9.5051, Z -2.1667, A 0.000, B 0.000, C 0.000 }
gfCNCPoint1[22036] = {X 273.4964, Y 9.5051, Z -2.1667, A 0.000, B 0.000, C 0.000 }
gfCNCPoint1[22037] = {X 273.7797, Y 10.3731, Z -2.1667, A 0.000, B 0.000, C 0.000 }
gfCNCPoint1[22038] = {X 273.9521, Y 11.2698, Z -2.1667, A 0.000, B 0.000, C 0.000 }
gfCNCPoint1[22039] = {X 274.0110, Y 12.1809, Z -2.1667, A 0.000, B 0.000, C 0.000 }
gfCNCPoint1[22040] = {X 274.0106, Y 13.0529, Z -2.1667, A 0.000, B 0.000, C 0.000 }
gfCNCPoint1[22041] = {X 273.9421, Y 13.9776, Z -2.1667, A 0.000, B 0.000, C 0.000 }
gfCNCPoint1[22042] = {X 273.7565, Y 14.8861, Z -2.1667, A 0.000, B 0.000, C 0.000 }
gfCNCPoint1[22043] = {X 273.4570, Y 15.7637, Z -2.1667, A 0.000, B 0.000, C 0.000 }
gfCNCPoint1[22044] = {X 271.2396, Y 14.8453, Z -2.1667, A 0.000, B 0.000, C 0.000 }
gfCNCPoint1[22045] = {X 270.7501, Y 15.7460, Z -2.1667, A 0.000, B 0.000, C 0.000 }
gfCNCPoint1[22046] = {X 270.0831, Y 16.5245, Z -2.1667, A 0.000, B 0.000, C 0.000 }
gfCNCPoint1[22047] = {X 270.0829, Y 40.6621, Z -2.1667, A 0.000, B 0.000, C 0.000 }
gfCNCPoint1[22048] = {X 270.7238, Y 41.4030, Z -2.1667, A 0.000, B 0.000, C 0.000 }
gfCNCPoint1[22049] = {X 271.2037, Y 42.2570, Z -2.1667, A 0.000, B 0.000, C 0.000 }
gfCNCPoint1[22050] = {X 271.5034, Y 43.1896, Z -2.1667, A 0.000, B 0.000, C 0.000 }
gfCNCPoint1[22051] = {X 271.6108, Y 44.1633, Z -2.1667, A 0.000, B 0.000, C 0.000 }
gfCNCPoint1[22052] = {X 271.6110, Y 45.0000, Z -2.1667, A 0.000, B 0.000, C 0.000 }
gfCNCPoint1[22053] = {X 271.5959, Y 45.3844, Z -2.1667, A 0.000, B 0.000, C 0.000 }
gfCNCPoint1[22054] = {X 271.5505, Y 45.7664, Z -2.1667, A 0.000, B 0.000, C 0.000 }
gfCNCPoint1[22055] = {X 271.2989, Y 46.7171, Z -2.1667, A 0.000, B 0.000, C 0.000 }
gfCNCPoint1[22056] = {X 270.8619, Y 47.5982, Z -2.1667, A 0.000, B 0.000, C 0.000 }
gfCNCPoint1[22057] = {X 270.2571, Y 48.3736, Z -2.1667, A 0.000, B 0.000, C 0.000 }
gfCNCPoint1[22058] = {X 269.5090, Y 49.0121, Z -2.1667, A 0.000, B 0.000, C 0.000 }
gfCNCPoint1[22059] = {X 268.6482, Y 49.4876, Z -2.1667, A 0.000, B 0.000, C 0.000 }
gfCNCPoint1[22060] = {X 267.7095, Y 49.7809, Z -2.1667, A 0.000, B 0.000, C 0.000 }
gfCNCPoint1[22061] = {X 266.7310, Y 49.8800, Z -2.1667, A 0.000, B 0.000, C 0.000 }
gfCNCPoint1[22062] = {X 262.1384, Y 49.8800, Z -2.1667, A 0.000, B 0.000, C 0.000 }
gfCNCPoint1[22063] = {X 262.1384, Y 54.6800, Z -2.1667, A 0.000, B 0.000, C 0.000 }
gfCNCPoint1[22064] = {X 260.2788, Y 54.6800, Z -2.1667, A 0.000, B 0.000, C 0.000 }
gfCNCPoint1[22065] = {X 261.9952, Y 55.3610, Z -2.1667, A 0.000, B 0.000, C 0.000 }
gfCNCPoint1[22066] = {X 262.0627, Y 55.0197, Z -2.1667, A 0.000, B 0.000, C 0.000 }
gfCNCPoint1[22067] = {X 262.1384, Y 54.6800, Z -2.1667, A 0.000, B 0.000, C 0.000 }
gfCNCPoint1[22068] = {X 262.1384, Y 52.2800, Z -2.1667, A 0.000, B 0.000, C 0.000 }
gfCNCPoint1[22069] = {X 260.2810, Y 52.2800, Z -2.1667, A 0.000, B 0.000, C 0.000 }
gfCNCPoint1[22070] = {X 259.1879, Y 52.1965, Z -2.1667, A 0.000, B 0.000, C 0.000 }
gfCNCPoint1[22071] = {X 258.1198, Y 51.9498, Z -2.1667, A 0.000, B 0.000, C 0.000 }
gfCNCPoint1[22072] = {X 257.1008, Y 51.5455, Z -2.1667, A 0.000, B 0.000, C 0.000 }
gfCNCPoint1[22073] = {X 256.1541, Y 50.9927, Z -2.1667, A 0.000, B 0.000, C 0.000 }
gfCNCPoint1[22074] = {X 255.3011, Y 50.3041, Z -2.1667, A 0.000, B 0.000, C 0.000 }
gfCNCPoint1[22075] = {X 253.6573, Y 52.0528, Z -2.1667, A 0.000, B 0.000, C 0.000 }
gfCNCPoint1[22076] = {X 253.4971, Y 51.8987, Z -2.1667, A 0.000, B 0.000, C 0.000 }
gfCNCPoint1[22077] = {X 253.3406, Y 51.7410, Z -2.1667, A 0.000, B 0.000, C 0.000 }
gfCNCPoint1[22078] = {X 253.2748, Y 51.8082, Z -2.1667, A 0.000, B 0.000, C 0.000 }
gfCNCPoint1[22079] = {X 253.2084, Y 51.8747, Z -2.1667, A 0.000, B 0.000, C 0.000 }
gfCNCPoint1[22080] = {X 253.6573, Y 52.0528, Z -2.1667, A 0.000, B 0.000, C 0.000 }
gfCNCPoint1[22081] = {X 255.3011, Y 50.3041, Z -2.1667, A 0.000, B 0.000, C 0.000 }
gfCNCPoint1[22082] = {X 255.1807, Y 50.1883, Z -2.1667, A 0.000, B 0.000, C 0.000 }
gfCNCPoint1[22083] = {X 255.0630, Y 50.0697, Z -2.1667, A 0.000, B 0.000, C 0.000 }
gfCNCPoint1[22084] = {X 254.3405, Y 49.1989, Z -2.1667, A 0.000, B 0.000, C 0.000 }
gfCNCPoint1[22085] = {X 253.7617, Y 48.2267, Z -2.1667, A 0.000, B 0.000, C 0.000 }
gfCNCPoint1[22086] = {X 253.3406, Y 47.1766, Z -2.1667, A 0.000, B 0.000, C 0.000 }
gfCNCPoint1[22087] = {X 252.9194, Y 48.2267, Z -2.1667, A 0.000, B 0.000, C 0.000 }
gfCNCPoint1[22088] = {X 252.3406, Y 49.1989, Z -2.1667, A 0.000, B 0.000, C 0.000 }
gfCNCPoint1[22089] = {X 251.6182, Y 50.0697, Z -2.1667, A 0.000, B 0.000, C 0.000 }
gfCNCPoint1[22090] = {X 251.5687, Y 50.1202, Z -2.1667, A 0.000, B 0.000, C 0.000 }
gfCNCPoint1[22091] = {X 251.5187, Y 50.1702, Z -2.1667, A 0.000, B 0.000, C 0.000 }
gfCNCPoint1[22092] = {X 250.7132, Y 50.8600, Z -2.1667, A 0.000, B 0.000, C 0.000 }
gfCNCPoint1[22093] = {X 249.8159, Y 51.4254, Z -2.1667, A 0.000, B 0.000, C 0.000 }
gfCNCPoint1[22094] = {X 248.8460, Y 51.8545, Z -2.1667, A 0.000, B 0.000, C 0.000 }
gfCNCPoint1[22095] = {X 247.8241, Y 52.1381, Z -2.1667, A 0.000, B 0.000, C 0.000 }
gfCNCPoint1[22096] = {X 247.8930, Y 52.2640, Z -2.1667, A 0.000, B 0.000, C 0.000 }
gfCNCPoint1[22097] = {X 247.9604, Y 52.3908, Z -2.1667, A 0.000, B 0.000, C 0.000 }
gfCNCPoint1[22098] = {X 250.3413, Y 53.3191, Z -2.1667, A 0.000, B 0.000, C 0.000 }
gfCNCPoint1[22099] = {X 264.1528, Y 58.7991, Z -2.1667, A 0.000, B 0.000, C 0.000 }
gfCNCPoint1[22100] = {X 264.1527, Y 58.0000, Z -2.1667, A 0.000, B 0.000, C 0.000 }
gfCNCPoint1[22101] = {X 264.2034, Y 56.8946, Z -2.1667, A 0.000, B 0.000, C 0.000 }
gfCNCPoint1[22102] = {X 264.3550, Y 55.7984, Z -2.1667, A 0.000, B 0.000, C 0.000 }
gfCNCPoint1[22103] = {X 264.4113, Y 55.5136, Z -2.1667, A 0.000, B 0.000, C 0.000 }
gfCNCPoint1[22104] = {X 264.4745, Y 55.2303, Z -2.1667, A 0.000, B 0.000, C 0.000 }
gfCNCPoint1[22105] = {X 264.9369, Y 53.7185, Z -2.1667, A 0.000, B 0.000, C 0.000 }
gfCNCPoint1[22106] = {X 265.5928, Y 52.2800, Z -2.1667, A 0.000, B 0.000, C 0.000 }
gfCNCPoint1[22107] = {X 262.1384, Y 52.2800, Z -2.1667, A 0.000, B 0.000, C 0.000 }
gfCNCPoint1[22108] = {X 262.1384, Y 49.8800, Z -2.1667, A 0.000, B 0.000, C 0.000 }
gfCNCPoint1[22109] = {X 260.2876, Y 49.8800, Z -2.1667, A 0.000, B 0.000, C 0.000 }
gfCNCPoint1[22110] = {X 259.2646, Y 49.7716, Z -2.1667, A 0.000, B 0.000, C 0.000 }
gfCNCPoint1[22111] = {X 258.2870, Y 49.4511, Z -2.1667, A 0.000, B 0.000, C 0.000 }
gfCNCPoint1[22112] = {X 257.3984, Y 48.9328, Z -2.1667, A 0.000, B 0.000, C 0.000 }
gfCNCPoint1[22113] = {X 256.6382, Y 48.2398, Z -2.1667, A 0.000, B 0.000, C 0.000 }
gfCNCPoint1[22114] = {X 256.0401, Y 47.4028, Z -2.1667, A 0.000, B 0.000, C 0.000 }
gfCNCPoint1[22115] = {X 255.6308, Y 46.4590, Z -2.1667, A 0.000, B 0.000, C 0.000 }
gfCNCPoint1[22116] = {X 255.4666, Y 45.7568, Z -2.1667, A 0.000, B 0.000, C 0.000 }
gfCNCPoint1[22117] = {X 255.4077, Y 45.0380, Z -2.1667, A 0.000, B 0.000, C 0.000 }
gfCNCPoint1[22118] = {X 255.4080, Y 44.1417, Z -2.1667, A 0.000, B 0.000, C 0.000 }
gfCNCPoint1[22119] = {X 255.5183, Y 43.1751, Z -2.1667, A 0.000, B 0.000, C 0.000 }
gfCNCPoint1[22120] = {X 255.8181, Y 42.2497, Z -2.1667, A 0.000, B 0.000, C 0.000 }
gfCNCPoint1[22121] = {X 256.2955, Y 41.4021, Z -2.1667, A 0.000, B 0.000, C 0.000 }
gfCNCPoint1[22122] = {X 256.9315, Y 40.6660, Z -2.1667, A 0.000, B 0.000, C 0.000 }
gfCNCPoint1[22123] = {X 256.9315, Y 35.0338, Z -2.1667, A 0.000, B 0.000, C 0.000 }
gfCNCPoint1[22124] = {X 255.1088, Y 35.0338, Z -2.1667, A 0.000, B 0.000, C 0.000 }
gfCNCPoint1[22125] = {X 251.0863, Y 42.8701, Z -2.1667, A 0.000, B 0.000, C 0.000 }
gfCNCPoint1[22126] = {X 251.2236, Y 43.5125, Z -2.1667, A 0.000, B 0.000, C 0.000 }
gfCNCPoint1[22127] = {X 251.2734, Y 44.1675, Z -2.1667, A 0.000, B 0.000, C 0.000 }
gfCNCPoint1[22128] = {X 251.2736, Y 45.0000, Z -2.1667, A 0.000, B 0.000, C 0.000 }
gfCNCPoint1[22129] = {X 251.2174, Y 45.7380, Z -2.1667, A 0.000, B 0.000, C 0.000 }
gfCNCPoint1[22130] = {X 251.0503, Y 46.4590, Z -2.1667, A 0.000, B 0.000, C 0.000 }
gfCNCPoint1[22131] = {X 250.6346, Y 47.4142, Z -2.1667, A 0.000, B 0.000, C 0.000 }
gfCNCPoint1[22132] = {X 250.0255, Y 48.2593, Z -2.1667, A 0.000, B 0.000, C 0.000 }
gfCNCPoint1[22133] = {X 249.2510, Y 48.9560, Z -2.1667, A 0.000, B 0.000, C 0.000 }
gfCNCPoint1[22134] = {X 248.3462, Y 49.4723, Z -2.1667, A 0.000, B 0.000, C 0.000 }
gfCNCPoint1[22135] = {X 247.3525, Y 49.7849, Z -2.1667, A 0.000, B 0.000, C 0.000 }
gfCNCPoint1[22136] = {X 246.8754, Y 49.8562, Z -2.1667, A 0.000, B 0.000, C 0.000 }
gfCNCPoint1[22137] = {X 246.3936, Y 49.8800, Z -2.1667, A 0.000, B 0.000, C 0.000 }
gfCNCPoint1[22138] = {X 242.5312, Y 49.8800, Z -2.1667, A 0.000, B 0.000, C 0.000 }
gfCNCPoint1[22139] = {X 242.5312, Y 49.4000, Z -2.1667, A 0.000, B 0.000, C 0.000 }
gfCNCPoint1[22140] = {X 239.8075, Y 49.4000, Z -2.1667, A 0.000, B 0.000, C 0.000 }
gfCNCPoint1[22141] = {X 238.8284, Y 49.2897, Z -2.1667, A 0.000, B 0.000, C 0.000 }
gfCNCPoint1[22142] = {X 237.8984, Y 48.9643, Z -2.1667, A 0.000, B 0.000, C 0.000 }
gfCNCPoint1[22143] = {X 237.0641, Y 48.4401, Z -2.1667, A 0.000, B 0.000, C 0.000 }
gfCNCPoint1[22144] = {X 236.3674, Y 47.7434, Z -2.1667, A 0.000, B 0.000, C 0.000 }
gfCNCPoint1[22145] = {X 235.8432, Y 46.9091, Z -2.1667, A 0.000, B 0.000, C 0.000 }
gfCNCPoint1[22146] = {X 235.5178, Y 45.9791, Z -2.1667, A 0.000, B 0.000, C 0.000 }
gfCNCPoint1[22147] = {X 235.4075, Y 45.0000, Z -2.1667, A 0.000, B 0.000, C 0.000 }
gfCNCPoint1[22148] = {X 235.4079, Y 44.1483, Z -2.1667, A 0.000, B 0.000, C 0.000 }
gfCNCPoint1[22149] = {X 235.5063, Y 43.2816, Z -2.1667, A 0.000, B 0.000, C 0.000 }
gfCNCPoint1[22150] = {X 235.7737, Y 42.4514, Z -2.1667, A 0.000, B 0.000, C 0.000 }
gfCNCPoint1[22151] = {X 236.1996, Y 41.6903, Z -2.1667, A 0.000, B 0.000, C 0.000 }
gfCNCPoint1[22152] = {X 236.7672, Y 41.0281, Z -2.1667, A 0.000, B 0.000, C 0.000 }
gfCNCPoint1[22153] = {X 237.4544, Y 40.4909, Z -2.1667, A 0.000, B 0.000, C 0.000 }
gfCNCPoint1[22154] = {X 238.2339, Y 40.0998, Z -2.1667, A 0.000, B 0.000, C 0.000 }
gfCNCPoint1[22155] = {X 242.1752, Y 32.3853, Z -2.1667, A 0.000, B 0.000, C 0.000 }
gfCNCPoint1[22156] = {X 241.0117, Y 31.5929, Z -2.1667, A 0.000, B 0.000, C 0.000 }
gfCNCPoint1[22157] = {X 239.9549, Y 30.6632, Z -2.1667, A 0.000, B 0.000, C 0.000 }
gfCNCPoint1[22158] = {X 239.0207, Y 29.6103, Z -2.1667, A 0.000, B 0.000, C 0.000 }
gfCNCPoint1[22159] = {X 238.2234, Y 28.4503, Z -2.1667, A 0.000, B 0.000, C 0.000 }
gfCNCPoint1[22160] = {X 237.5752, Y 27.2008, Z -2.1667, A 0.000, B 0.000, C 0.000 }
gfCNCPoint1[22161] = {X 237.0859, Y 25.8809, Z -2.1667, A 0.000, B 0.000, C 0.000 }
gfCNCPoint1[22162] = {X 236.6642, Y 24.0613, Z -2.1667, A 0.000, B 0.000, C 0.000 }
gfCNCPoint1[22163] = {X 236.4493, Y 22.2058, Z -2.1667, A 0.000, B 0.000, C 0.000 }
gfCNCPoint1[22164] = {X 236.4441, Y 20.3379, Z -2.1667, A 0.000, B 0.000, C 0.000 }
gfCNCPoint1[22165] = {X 236.6486, Y 18.4812, Z -2.1667, A 0.000, B 0.000, C 0.000 }
gfCNCPoint1[22166] = {X 237.0602, Y 16.6592, Z -2.1667, A 0.000, B 0.000, C 0.000 }
gfCNCPoint1[22167] = {X 237.6343, Y 15.0731, Z -2.1667, A 0.000, B 0.000, C 0.000 }
gfCNCPoint1[22168] = {X 238.4264, Y 13.5838, Z -2.1667, A 0.000, B 0.000, C 0.000 }
gfCNCPoint1[22169] = {X 239.4207, Y 12.2212, Z -2.1667, A 0.000, B 0.000, C 0.000 }
gfCNCPoint1[22170] = {X 240.5974, Y 11.0125, Z -2.1667, A 0.000, B 0.000, C 0.000 }
gfCNCPoint1[22171] = {X 241.9328, Y 9.9819, Z -2.1667, A 0.000, B 0.000, C 0.000 }
gfCNCPoint1[22172] = {X 243.4002, Y 9.1500, Z -2.1667, A 0.000, B 0.000, C 0.000 }
gfCNCPoint1[22173] = {X 244.9704, Y 8.5335, Z -2.1667, A 0.000, B 0.000, C 0.000 }
gfCNCPoint1[22174] = {X 246.6118, Y 8.1447, Z -2.1667, A 0.000, B 0.000, C 0.000 }
gfCNCPoint1[22175] = {X 248.7155, Y 7.8721, Z -2.1667, A 0.000, B 0.000, C 0.000 }
gfCNCPoint1[22176] = {X 250.8352, Y 7.7916, Z -2.1667, A 0.000, B 0.000, C 0.000 }
gfCNCPoint1[22177] = {X 266.7640, Y 7.7916, Z -2.1667, A 0.000, B 0.000, C 0.000 }
gfCNCPoint1[22178] = {X 267.7367, Y 7.9085, Z -2.1667, A 0.000, B 0.000, C 0.000 }
gfCNCPoint1[22179] = {X 268.6595, Y 8.2376, Z -2.1667, A 0.000, B 0.000, C 0.000 }
gfCNCPoint1[22180] = {X 269.4866, Y 8.7626, Z -2.1667, A 0.000, B 0.000, C 0.000 }
gfCNCPoint1[22181] = {X 270.1772, Y 9.4575, Z -2.1667, A 0.000, B 0.000, C 0.000 }
gfCNCPoint1[22182] = {X 270.6970, Y 10.2879, Z -2.1667, A 0.000, B 0.000, C 0.000 }
gfCNCPoint1[22183] = {X 271.0203, Y 11.2127, Z -2.1667, A 0.000, B 0.000, C 0.000 }
gfCNCPoint1[22184] = {X 271.1310, Y 12.1862, Z -2.1667, A 0.000, B 0.000, C 0.000 }
gfCNCPoint1[22185] = {X 271.1308, Y 13.0233, Z -2.1667, A 0.000, B 0.000, C 0.000 }
gfCNCPoint1[22186] = {X 271.0225, Y 13.9495, Z -2.1667, A 0.000, B 0.000, C 0.000 }
gfCNCPoint1[22187] = {X 270.7214, Y 14.8320, Z -2.1667, A 0.000, B 0.000, C 0.000 }
gfCNCPoint1[22188] = {X 270.2411, Y 15.6312, Z -2.1667, A 0.000, B 0.000, C 0.000 }
gfCNCPoint1[22189] = {X 269.6031, Y 16.3113, Z -2.1667, A 0.000, B 0.000, C 0.000 }
gfCNCPoint1[22190] = {X 269.6029, Y 40.8753, Z -2.1667, A 0.000, B 0.000, C 0.000 }
gfCNCPoint1[22191] = {X 270.2478, Y 41.5645, Z -2.1667, A 0.000, B 0.000, C 0.000 }
gfCNCPoint1[22192] = {X 270.7308, Y 42.3753, Z -2.1667, A 0.000, B 0.000, C 0.000 }
gfCNCPoint1[22193] = {X 271.0298, Y 43.2705, Z -2.1667, A 0.000, B 0.000, C 0.000 }
gfCNCPoint1[22194] = {X 271.1310, Y 44.2089, Z -2.1667, A 0.000, B 0.000, C 0.000 }
gfCNCPoint1[22195] = {X 271.1310, Y 45.0000, Z -2.1667, A 0.000, B 0.000, C 0.000 }
gfCNCPoint1[22196] = {X 271.0207, Y 45.9791, Z -2.1667, A 0.000, B 0.000, C 0.000 }
gfCNCPoint1[22197] = {X 270.6953, Y 46.9091, Z -2.1667, A 0.000, B 0.000, C 0.000 }
gfCNCPoint1[22198] = {X 270.1711, Y 47.7434, Z -2.1667, A 0.000, B 0.000, C 0.000 }
gfCNCPoint1[22199] = {X 269.4744, Y 48.4401, Z -2.1667, A 0.000, B 0.000, C 0.000 }
gfCNCPoint1[22200] = {X 268.6401, Y 48.9643, Z -2.1667, A 0.000, B 0.000, C 0.000 }
gfCNCPoint1[22201] = {X 267.7101, Y 49.2897, Z -2.1667, A 0.000, B 0.000, C 0.000 }
gfCNCPoint1[22202] = {X 266.7310, Y 49.4000, Z -2.1667, A 0.000, B 0.000, C 0.000 }
gfCNCPoint1[22203] = {X 260.2876, Y 49.4000, Z -2.1667, A 0.000, B 0.000, C 0.000 }
gfCNCPoint1[22204] = {X 259.3085, Y 49.2897, Z -2.1667, A 0.000, B 0.000, C 0.000 }
gfCNCPoint1[22205] = {X 258.3785, Y 48.9643, Z -2.1667, A 0.000, B 0.000, C 0.000 }
gfCNCPoint1[22206] = {X 257.5442, Y 48.4400, Z -2.1667, A 0.000, B 0.000, C 0.000 }
gfCNCPoint1[22207] = {X 256.8475, Y 47.7433, Z -2.1667, A 0.000, B 0.000, C 0.000 }
gfCNCPoint1[22208] = {X 256.3233, Y 46.9091, Z -2.1667, A 0.000, B 0.000, C 0.000 }
gfCNCPoint1[22209] = {X 255.9979, Y 45.9791, Z -2.1667, A 0.000, B 0.000, C 0.000 }
gfCNCPoint1[22210] = {X 255.8876, Y 45.0000, Z -2.1667, A 0.000, B 0.000, C 0.000 }
gfCNCPoint1[22211] = {X 255.8880, Y 44.1483, Z -2.1667, A 0.000, B 0.000, C 0.000 }
gfCNCPoint1[22212] = {X 255.9984, Y 43.2275, Z -2.1667, A 0.000, B 0.000, C 0.000 }
gfCNCPoint1[22213] = {X 256.2993, Y 42.3503, Z -2.1667, A 0.000, B 0.000, C 0.000 }
gfCNCPoint1[22214] = {X 256.7775, Y 41.5556, Z -2.1667, A 0.000, B 0.000, C 0.000 }
gfCNCPoint1[22215] = {X 257.4115, Y 40.8789, Z -2.1667, A 0.000, B 0.000, C 0.000 }
gfCNCPoint1[22216] = {X 257.4115, Y 34.5538, Z -2.1667, A 0.000, B 0.000, C 0.000 }
gfCNCPoint1[22217] = {X 254.8156, Y 34.5538, Z -2.1667, A 0.000, B 0.000, C 0.000 }
gfCNCPoint1[22218] = {X 250.5701, Y 42.8246, Z -2.1667, A 0.000, B 0.000, C 0.000 }
gfCNCPoint1[22219] = {X 250.7374, Y 43.5078, Z -2.1667, A 0.000, B 0.000, C 0.000 }
gfCNCPoint1[22220] = {X 250.7936, Y 44.2089, Z -2.1667, A 0.000, B 0.000, C 0.000 }
gfCNCPoint1[22221] = {X 250.7936, Y 45.0000, Z -2.1667, A 0.000, B 0.000, C 0.000 }
gfCNCPoint1[22222] = {X 250.6832, Y 45.9791, Z -2.1667, A 0.000, B 0.000, C 0.000 }
gfCNCPoint1[22223] = {X 250.3578, Y 46.9091, Z -2.1667, A 0.000, B 0.000, C 0.000 }
gfCNCPoint1[22224] = {X 249.8336, Y 47.7434, Z -2.1667, A 0.000, B 0.000, C 0.000 }
gfCNCPoint1[22225] = {X 249.1369, Y 48.4401, Z -2.1667, A 0.000, B 0.000, C 0.000 }
gfCNCPoint1[22226] = {X 248.3026, Y 48.9643, Z -2.1667, A 0.000, B 0.000, C 0.000 }
gfCNCPoint1[22227] = {X 247.3727, Y 49.2897, Z -2.1667, A 0.000, B 0.000, C 0.000 }
gfCNCPoint1[22228] = {X 246.3936, Y 49.4000, Z -2.1667, A 0.000, B 0.000, C 0.000 }
gfCNCPoint1[22229] = {X 242.5312, Y 49.4000, Z -2.1667, A 0.000, B 0.000, C 0.000 }
gfCNCPoint1[22230] = {X 242.5312, Y 49.8800, Z -2.1667, A 0.000, B 0.000, C 0.000 }
gfCNCPoint1[22231] = {X 243.4812, Y 50.5824, Z -2.1667, A 0.000, B 0.000, C 0.000 }
gfCNCPoint1[22232] = {X 244.3384, Y 51.3953, Z -2.1667, A 0.000, B 0.000, C 0.000 }
gfCNCPoint1[22233] = {X 245.0903, Y 52.3066, Z -2.1667, A 0.000, B 0.000, C 0.000 }
gfCNCPoint1[22234] = {X 245.7256, Y 53.3027, Z -2.1667, A 0.000, B 0.000, C 0.000 }
gfCNCPoint1[22235] = {X 245.9756, Y 53.7846, Z -2.1667, A 0.000, B 0.000, C 0.000 }
gfCNCPoint1[22236] = {X 246.1982, Y 54.2797, Z -2.1667, A 0.000, B 0.000, C 0.000 }
gfCNCPoint1[22237] = {X 249.4594, Y 55.5512, Z -2.1667, A 0.000, B 0.000, C 0.000 }
gfCNCPoint1[22238] = {X 267.2832, Y 62.6232, Z -2.1667, A 0.000, B 0.000, C 0.000 }
gfCNCPoint1[22239] = {X 266.8848, Y 61.4478, Z -2.1667, A 0.000, B 0.000, C 0.000 }
gfCNCPoint1[22240] = {X 266.6400, Y 60.2311, Z -2.1667, A 0.000, B 0.000, C 0.000 }
gfCNCPoint1[22241] = {X 266.5529, Y 58.9930, Z -2.1667, A 0.000, B 0.000, C 0.000 }
gfCNCPoint1[22242] = {X 266.5527, Y 58.0000, Z -2.1667, A 0.000, B 0.000, C 0.000 }
gfCNCPoint1[22243] = {X 266.6262, Y 56.8093, Z -2.1667, A 0.000, B 0.000, C 0.000 }
gfCNCPoint1[22244] = {X 266.8456, Y 55.6367, Z -2.1667, A 0.000, B 0.000, C 0.000 }
gfCNCPoint1[22245] = {X 267.2076, Y 54.5000, Z -2.1667, A 0.000, B 0.000, C 0.000 }
gfCNCPoint1[22246] = {X 267.7067, Y 53.4164, Z -2.1667, A 0.000, B 0.000, C 0.000 }
gfCNCPoint1[22247] = {X 268.4728, Y 52.2132, Z -2.1667, A 0.000, B 0.000, C 0.000 }
gfCNCPoint1[22248] = {X 269.4075, Y 51.1357, Z -2.1667, A 0.000, B 0.000, C 0.000 }
gfCNCPoint1[22249] = {X 270.4903, Y 50.2072, Z -2.1667, A 0.000, B 0.000, C 0.000 }
gfCNCPoint1[22250] = {X 271.6979, Y 49.4479, Z -2.1667, A 0.000, B 0.000, C 0.000 }
gfCNCPoint1[22251] = {X 273.0039, Y 48.8744, Z -2.1667, A 0.000, B 0.000, C 0.000 }
gfCNCPoint1[22252] = {X 274.3800, Y 48.4989, Z -2.1667, A 0.000, B 0.000, C 0.000 }
gfCNCPoint1[22253] = {X 275.3020, Y 48.3648, Z -2.1667, A 0.000, B 0.000, C 0.000 }
gfCNCPoint1[22254] = {X 276.2327, Y 48.3200, Z -2.1667, A 0.000, B 0.000, C 0.000 }
gfCNCPoint1[22255] = {X 281.0411, Y 48.3200, Z -2.1667, A 0.000, B 0.000, C 0.000 }
gfCNCPoint1[22256] = {X 280.4347, Y 47.5134, Z -2.1667, A 0.000, B 0.000, C 0.000 }
gfCNCPoint1[22257] = {X 280.0072, Y 46.5992, Z -2.1667, A 0.000, B 0.000, C 0.000 }
gfCNCPoint1[22258] = {X 279.7768, Y 45.6167, Z -2.1667, A 0.000, B 0.000, C 0.000 }
gfCNCPoint1[22259] = {X 279.7488, Y 45.3288, Z -2.1667, A 0.000, B 0.000, C 0.000 }
gfCNCPoint1[22260] = {X 279.7378, Y 45.0398, Z -2.1667, A 0.000, B 0.000, C 0.000 }
gfCNCPoint1[22261] = {X 279.7377, Y 44.2037, Z -2.1667, A 0.000, B 0.000, C 0.000 }
gfCNCPoint1[22262] = {X 279.8426, Y 43.2204, Z -2.1667, A 0.000, B 0.000, C 0.000 }
gfCNCPoint1[22263] = {X 280.1416, Y 42.2777, Z -2.1667, A 0.000, B 0.000, C 0.000 }
gfCNCPoint1[22264] = {X 280.6226, Y 41.4137, Z -2.1667, A 0.000, B 0.000, C 0.000 }
gfCNCPoint1[22265] = {X 281.2662, Y 40.6629, Z -2.1667, A 0.000, B 0.000, C 0.000 }
gfCNCPoint1[22266] = {X 281.2658, Y 16.5248, Z -2.1667, A 0.000, B 0.000, C 0.000 }
gfCNCPoint1[22267] = {X 280.6244, Y 15.7831, Z -2.1667, A 0.000, B 0.000, C 0.000 }
gfCNCPoint1[22268] = {X 280.1443, Y 14.9281, Z -2.1667, A 0.000, B 0.000, C 0.000 }
gfCNCPoint1[22269] = {X 279.8447, Y 13.9945, Z -2.1667, A 0.000, B 0.000, C 0.000 }
gfCNCPoint1[22270] = {X 279.7378, Y 13.0198, Z -2.1667, A 0.000, B 0.000, C 0.000 }
gfCNCPoint1[22271] = {X 279.7377, Y 12.1868, Z -2.1667, A 0.000, B 0.000, C 0.000 }
gfCNCPoint1[22272] = {X 279.8242, Y 11.2718, Z -2.1667, A 0.000, B 0.000, C 0.000 }
gfCNCPoint1[22273] = {X 280.0808, Y 10.3892, Z -2.1667, A 0.000, B 0.000, C 0.000 }
gfCNCPoint1[22274] = {X 280.5255, Y 9.5281, Z -2.1667, A 0.000, B 0.000, C 0.000 }
gfCNCPoint1[22275] = {X 281.1316, Y 8.7718, Z -2.1667, A 0.000, B 0.000, C 0.000 }
gfCNCPoint1[22276] = {X 281.8752, Y 8.1503, Z -2.1667, A 0.000, B 0.000, C 0.000 }
gfCNCPoint1[22277] = {X 282.7270, Y 7.6880, Z -2.1667, A 0.000, B 0.000, C 0.000 }
gfCNCPoint1[22278] = {X 283.6533, Y 7.4030, Z -2.1667, A 0.000, B 0.000, C 0.000 }
gfCNCPoint1[22279] = {X 284.6177, Y 7.3068, Z -2.1667, A 0.000, B 0.000, C 0.000 }
gfCNCPoint1[22280] = {X 291.0611, Y 7.3068, Z -2.1667, A 0.000, B 0.000, C 0.000 }
gfCNCPoint1[22281] = {X 292.0255, Y 7.4030, Z -2.1667, A 0.000, B 0.000, C 0.000 }
gfCNCPoint1[22282] = {X 292.9518, Y 7.6880, Z -2.1667, A 0.000, B 0.000, C 0.000 }
gfCNCPoint1[22283] = {X 293.8036, Y 8.1503, Z -2.1667, A 0.000, B 0.000, C 0.000 }
gfCNCPoint1[22284] = {X 294.5472, Y 8.7718, Z -2.1667, A 0.000, B 0.000, C 0.000 }
gfCNCPoint1[22285] = {X 295.1533, Y 9.5281, Z -2.1667, A 0.000, B 0.000, C 0.000 }
gfCNCPoint1[22286] = {X 295.5980, Y 10.3892, Z -2.1667, A 0.000, B 0.000, C 0.000 }
gfCNCPoint1[22287] = {X 295.8044, Y 11.0397, Z -2.1667, A 0.000, B 0.000, C 0.000 }
gfCNCPoint1[22288] = {X 295.9180, Y 11.7127, Z -2.1667, A 0.000, B 0.000, C 0.000 }
gfCNCPoint1[22289] = {X 295.9354, Y 11.9495, Z -2.1667, A 0.000, B 0.000, C 0.000 }
gfCNCPoint1[22290] = {X 295.9411, Y 12.1868, Z -2.1667, A 0.000, B 0.000, C 0.000 }
gfCNCPoint1[22291] = {X 295.9409, Y 13.0237, Z -2.1667, A 0.000, B 0.000, C 0.000 }
gfCNCPoint1[22292] = {X 295.9342, Y 13.2382, Z -2.1667, A 0.000, B 0.000, C 0.000 }
gfCNCPoint1[22293] = {X 295.9180, Y 13.4521, Z -2.1667, A 0.000, B 0.000, C 0.000 }
gfCNCPoint1[22294] = {X 298.3067, Y 13.6853, Z -2.1667, A 0.000, B 0.000, C 0.000 }
gfCNCPoint1[22295] = {X 298.1360, Y 14.6939, Z -2.1667, A 0.000, B 0.000, C 0.000 }
gfCNCPoint1[22296] = {X 297.8256, Y 15.6687, Z -2.1667, A 0.000, B 0.000, C 0.000 }
gfCNCPoint1[22297] = {X 297.3817, Y 16.5904, Z -2.1667, A 0.000, B 0.000, C 0.000 }
gfCNCPoint1[22298] = {X 296.8129, Y 17.4407, Z -2.1667, A 0.000, B 0.000, C 0.000 }
gfCNCPoint1[22299] = {X 296.8133, Y 19.2365, Z -2.1667, A 0.000, B 0.000, C 0.000 }
gfCNCPoint1[22300] = {X 299.8000, Y 19.2365, Z -2.1667, A 0.000, B 0.000, C 0.000 }
gfCNCPoint1[22301] = {X 299.8002, Y 17.4403, Z -2.1667, A 0.000, B 0.000, C 0.000 }
gfCNCPoint1[22302] = {X 299.2315, Y 16.5901, Z -2.1667, A 0.000, B 0.000, C 0.000 }
gfCNCPoint1[22303] = {X 298.7877, Y 15.6685, Z -2.1667, A 0.000, B 0.000, C 0.000 }
gfCNCPoint1[22304] = {X 298.4773, Y 14.6938, Z -2.1667, A 0.000, B 0.000, C 0.000 }
gfCNCPoint1[22305] = {X 298.3067, Y 13.6853, Z -2.1667, A 0.000, B 0.000, C 0.000 }
gfCNCPoint1[22306] = {X 295.9180, Y 13.4521, Z -2.1667, A 0.000, B 0.000, C 0.000 }
gfCNCPoint1[22307] = {X 295.7559, Y 14.3098, Z -2.1667, A 0.000, B 0.000, C 0.000 }
gfCNCPoint1[22308] = {X 295.4436, Y 15.1248, Z -2.1667, A 0.000, B 0.000, C 0.000 }
gfCNCPoint1[22309] = {X 294.9910, Y 15.8712, Z -2.1667, A 0.000, B 0.000, C 0.000 }
gfCNCPoint1[22310] = {X 294.4127, Y 16.5250, Z -2.1667, A 0.000, B 0.000, C 0.000 }
gfCNCPoint1[22311] = {X 294.4139, Y 21.6365, Z -2.1667, A 0.000, B 0.000, C 0.000 }
gfCNCPoint1[22312] = {X 302.1997, Y 21.6365, Z -2.1667, A 0.000, B 0.000, C 0.000 }
gfCNCPoint1[22313] = {X 302.2003, Y 16.5247, Z -2.1667, A 0.000, B 0.000, C 0.000 }
gfCNCPoint1[22314] = {X 301.6222, Y 15.8709, Z -2.1667, A 0.000, B 0.000, C 0.000 }
gfCNCPoint1[22315] = {X 301.1697, Y 15.1246, Z -2.1667, A 0.000, B 0.000, C 0.000 }
gfCNCPoint1[22316] = {X 300.8575, Y 14.3096, Z -2.1667, A 0.000, B 0.000, C 0.000 }
gfCNCPoint1[22317] = {X 300.6953, Y 13.4521, Z -2.1667, A 0.000, B 0.000, C 0.000 }
gfCNCPoint1[22318] = {X 300.6791, Y 13.2371, Z -2.1667, A 0.000, B 0.000, C 0.000 }
gfCNCPoint1[22319] = {X 300.6724, Y 13.0215, Z -2.1667, A 0.000, B 0.000, C 0.000 }
gfCNCPoint1[22320] = {X 300.6723, Y 12.1868, Z -2.1667, A 0.000, B 0.000, C 0.000 }
gfCNCPoint1[22321] = {X 300.6780, Y 11.9495, Z -2.1667, A 0.000, B 0.000, C 0.000 }
gfCNCPoint1[22322] = {X 300.6953, Y 11.7127, Z -2.1667, A 0.000, B 0.000, C 0.000 }
gfCNCPoint1[22323] = {X 300.8090, Y 11.0397, Z -2.1667, A 0.000, B 0.000, C 0.000 }
gfCNCPoint1[22324] = {X 301.0154, Y 10.3892, Z -2.1667, A 0.000, B 0.000, C 0.000 }
gfCNCPoint1[22325] = {X 301.4601, Y 9.5281, Z -2.1667, A 0.000, B 0.000, C 0.000 }
gfCNCPoint1[22326] = {X 302.0662, Y 8.7718, Z -2.1667, A 0.000, B 0.000, C 0.000 }
gfCNCPoint1[22327] = {X 302.8098, Y 8.1503, Z -2.1667, A 0.000, B 0.000, C 0.000 }
gfCNCPoint1[22328] = {X 303.6616, Y 7.6880, Z -2.1667, A 0.000, B 0.000, C 0.000 }
gfCNCPoint1[22329] = {X 304.5879, Y 7.4030, Z -2.1667, A 0.000, B 0.000, C 0.000 }
gfCNCPoint1[22330] = {X 305.5523, Y 7.3068, Z -2.1667, A 0.000, B 0.000, C 0.000 }
gfCNCPoint1[22331] = {X 311.9957, Y 7.3068, Z -2.1667, A 0.000, B 0.000, C 0.000 }
gfCNCPoint1[22332] = {X 312.9478, Y 7.4006, Z -2.1667, A 0.000, B 0.000, C 0.000 }
gfCNCPoint1[22333] = {X 313.8632, Y 7.6783, Z -2.1667, A 0.000, B 0.000, C 0.000 }
gfCNCPoint1[22334] = {X 314.7069, Y 8.1292, Z -2.1667, A 0.000, B 0.000, C 0.000 }
gfCNCPoint1[22335] = {X 315.4464, Y 8.7361, Z -2.1667, A 0.000, B 0.000, C 0.000 }
gfCNCPoint1[22336] = {X 316.0533, Y 9.4756, Z -2.1667, A 0.000, B 0.000, C 0.000 }
gfCNCPoint1[22337] = {X 316.5043, Y 10.3193, Z -2.1667, A 0.000, B 0.000, C 0.000 }
gfCNCPoint1[22338] = {X 316.7820, Y 11.2348, Z -2.1667, A 0.000, B 0.000, C 0.000 }
gfCNCPoint1[22339] = {X 316.8757, Y 12.1868, Z -2.1667, A 0.000, B 0.000, C 0.000 }
gfCNCPoint1[22340] = {X 316.8755, Y 13.0237, Z -2.1667, A 0.000, B 0.000, C 0.000 }
gfCNCPoint1[22341] = {X 316.7681, Y 13.9974, Z -2.1667, A 0.000, B 0.000, C 0.000 }
gfCNCPoint1[22342] = {X 316.4683, Y 14.9300, Z -2.1667, A 0.000, B 0.000, C 0.000 }
gfCNCPoint1[22343] = {X 315.9883, Y 15.7840, Z -2.1667, A 0.000, B 0.000, C 0.000 }
gfCNCPoint1[22344] = {X 315.3474, Y 16.5249, Z -2.1667, A 0.000, B 0.000, C 0.000 }
gfCNCPoint1[22345] = {X 315.3472, Y 40.6617, Z -2.1667, A 0.000, B 0.000, C 0.000 }
gfCNCPoint1[22346] = {X 315.9886, Y 41.4033, Z -2.1667, A 0.000, B 0.000, C 0.000 }
gfCNCPoint1[22347] = {X 316.4689, Y 42.2581, Z -2.1667, A 0.000, B 0.000, C 0.000 }
gfCNCPoint1[22348] = {X 316.7686, Y 43.1917, Z -2.1667, A 0.000, B 0.000, C 0.000 }
gfCNCPoint1[22349] = {X 316.8755, Y 44.1664, Z -2.1667, A 0.000, B 0.000, C 0.000 }
gfCNCPoint1[22350] = {X 316.8757, Y 45.0000, Z -2.1667, A 0.000, B 0.000, C 0.000 }
gfCNCPoint1[22351] = {X 316.8749, Y 45.0899, Z -2.1667, A 0.000, B 0.000, C 0.000 }
gfCNCPoint1[22352] = {X 316.8724, Y 45.1799, Z -2.1667, A 0.000, B 0.000, C 0.000 }
gfCNCPoint1[22353] = {X 316.8594, Y 45.3987, Z -2.1667, A 0.000, B 0.000, C 0.000 }
gfCNCPoint1[22354] = {X 316.8366, Y 45.6167, Z -2.1667, A 0.000, B 0.000, C 0.000 }
gfCNCPoint1[22355] = {X 316.6062, Y 46.5992, Z -2.1667, A 0.000, B 0.000, C 0.000 }
gfCNCPoint1[22356] = {X 316.1787, Y 47.5134, Z -2.1667, A 0.000, B 0.000, C 0.000 }
gfCNCPoint1[22357] = {X 315.5723, Y 48.3200, Z -2.1667, A 0.000, B 0.000, C 0.000 }
gfCNCPoint1[22358] = {X 315.2205, Y 47.9934, Z -2.1667, A 0.000, B 0.000, C 0.000 }
gfCNCPoint1[22359] = {X 314.5413, Y 48.5889, Z -2.1667, A 0.000, B 0.000, C 0.000 }
gfCNCPoint1[22360] = {X 313.7548, Y 49.0331, Z -2.1667, A 0.000, B 0.000, C 0.000 }
gfCNCPoint1[22361] = {X 312.8942, Y 49.3073, Z -2.1667, A 0.000, B 0.000, C 0.000 }
gfCNCPoint1[22362] = {X 311.9957, Y 49.4000, Z -2.1667, A 0.000, B 0.000, C 0.000 }
gfCNCPoint1[22363] = {X 305.5523, Y 49.4000, Z -2.1667, A 0.000, B 0.000, C 0.000 }
gfCNCPoint1[22364] = {X 304.5732, Y 49.2897, Z -2.1667, A 0.000, B 0.000, C 0.000 }
gfCNCPoint1[22365] = {X 303.6432, Y 48.9643, Z -2.1667, A 0.000, B 0.000, C 0.000 }
gfCNCPoint1[22366] = {X 302.8089, Y 48.4400, Z -2.1667, A 0.000, B 0.000, C 0.000 }
gfCNCPoint1[22367] = {X 302.1122, Y 47.7433, Z -2.1667, A 0.000, B 0.000, C 0.000 }
gfCNCPoint1[22368] = {X 301.5880, Y 46.9091, Z -2.1667, A 0.000, B 0.000, C 0.000 }
gfCNCPoint1[22369] = {X 301.2626, Y 45.9791, Z -2.1667, A 0.000, B 0.000, C 0.000 }
gfCNCPoint1[22370] = {X 301.1523, Y 45.0000, Z -2.1667, A 0.000, B 0.000, C 0.000 }
gfCNCPoint1[22371] = {X 301.1524, Y 44.1991, Z -2.1667, A 0.000, B 0.000, C 0.000 }
gfCNCPoint1[22372] = {X 301.2705, Y 43.2557, Z -2.1667, A 0.000, B 0.000, C 0.000 }
gfCNCPoint1[22373] = {X 301.5738, Y 42.3546, Z -2.1667, A 0.000, B 0.000, C 0.000 }
gfCNCPoint1[22374] = {X 302.0502, Y 41.5318, Z -2.1667, A 0.000, B 0.000, C 0.000 }
gfCNCPoint1[22375] = {X 302.6807, Y 40.8202, Z -2.1667, A 0.000, B 0.000, C 0.000 }
gfCNCPoint1[22376] = {X 302.6807, Y 34.1143, Z -2.1667, A 0.000, B 0.000, C 0.000 }
gfCNCPoint1[22377] = {X 293.9337, Y 34.1143, Z -2.1667, A 0.000, B 0.000, C 0.000 }
gfCNCPoint1[22378] = {X 293.9328, Y 40.8664, Z -2.1667, A 0.000, B 0.000, C 0.000 }
gfCNCPoint1[22379] = {X 294.5727, Y 41.5614, Z -2.1667, A 0.000, B 0.000, C 0.000 }
gfCNCPoint1[22380] = {X 295.0536, Y 42.3746, Z -2.1667, A 0.000, B 0.000, C 0.000 }
gfCNCPoint1[22381] = {X 295.3541, Y 43.2703, Z -2.1667, A 0.000, B 0.000, C 0.000 }
gfCNCPoint1[22382] = {X 295.4611, Y 44.2089, Z -2.1667, A 0.000, B 0.000, C 0.000 }
gfCNCPoint1[22383] = {X 295.4611, Y 45.0000, Z -2.1667, A 0.000, B 0.000, C 0.000 }
gfCNCPoint1[22384] = {X 295.3508, Y 45.9791, Z -2.1667, A 0.000, B 0.000, C 0.000 }
gfCNCPoint1[22385] = {X 295.0254, Y 46.9091, Z -2.1667, A 0.000, B 0.000, C 0.000 }
gfCNCPoint1[22386] = {X 294.5012, Y 47.7434, Z -2.1667, A 0.000, B 0.000, C 0.000 }
gfCNCPoint1[22387] = {X 293.8045, Y 48.4401, Z -2.1667, A 0.000, B 0.000, C 0.000 }
gfCNCPoint1[22388] = {X 292.9702, Y 48.9643, Z -2.1667, A 0.000, B 0.000, C 0.000 }
gfCNCPoint1[22389] = {X 292.0402, Y 49.2897, Z -2.1667, A 0.000, B 0.000, C 0.000 }
gfCNCPoint1[22390] = {X 291.0611, Y 49.4000, Z -2.1667, A 0.000, B 0.000, C 0.000 }
gfCNCPoint1[22391] = {X 284.6177, Y 49.4000, Z -2.1667, A 0.000, B 0.000, C 0.000 }
gfCNCPoint1[22392] = {X 283.6386, Y 49.2897, Z -2.1667, A 0.000, B 0.000, C 0.000 }
gfCNCPoint1[22393] = {X 282.7086, Y 48.9643, Z -2.1667, A 0.000, B 0.000, C 0.000 }
gfCNCPoint1[22394] = {X 281.8743, Y 48.4400, Z -2.1667, A 0.000, B 0.000, C 0.000 }
gfCNCPoint1[22395] = {X 281.1776, Y 47.7433, Z -2.1667, A 0.000, B 0.000, C 0.000 }
gfCNCPoint1[22396] = {X 280.6534, Y 46.9091, Z -2.1667, A 0.000, B 0.000, C 0.000 }
gfCNCPoint1[22397] = {X 280.3280, Y 45.9791, Z -2.1667, A 0.000, B 0.000, C 0.000 }
gfCNCPoint1[22398] = {X 280.2177, Y 45.0000, Z -2.1667, A 0.000, B 0.000, C 0.000 }
gfCNCPoint1[22399] = {X 280.2177, Y 44.2065, Z -2.1667, A 0.000, B 0.000, C 0.000 }
gfCNCPoint1[22400] = {X 280.3230, Y 43.2697, Z -2.1667, A 0.000, B 0.000, C 0.000 }
gfCNCPoint1[22401] = {X 280.6232, Y 42.3760, Z -2.1667, A 0.000, B 0.000, C 0.000 }
gfCNCPoint1[22402] = {X 281.1048, Y 41.5656, Z -2.1667, A 0.000, B 0.000, C 0.000 }
gfCNCPoint1[22403] = {X 281.7462, Y 40.8747, Z -2.1667, A 0.000, B 0.000, C 0.000 }
gfCNCPoint1[22404] = {X 281.7458, Y 16.3116, Z -2.1667, A 0.000, B 0.000, C 0.000 }
gfCNCPoint1[22405] = {X 281.1009, Y 15.6224, Z -2.1667, A 0.000, B 0.000, C 0.000 }
gfCNCPoint1[22406] = {X 280.6179, Y 14.8115, Z -2.1667, A 0.000, B 0.000, C 0.000 }
gfCNCPoint1[22407] = {X 280.3189, Y 13.9163, Z -2.1667, A 0.000, B 0.000, C 0.000 }
gfCNCPoint1[22408] = {X 280.2177, Y 12.9779, Z -2.1667, A 0.000, B 0.000, C 0.000 }
gfCNCPoint1[22409] = {X 280.2177, Y 12.1868, Z -2.1667, A 0.000, B 0.000, C 0.000 }
gfCNCPoint1[22410] = {X 280.3280, Y 11.2077, Z -2.1667, A 0.000, B 0.000, C 0.000 }
gfCNCPoint1[22411] = {X 280.6534, Y 10.2777, Z -2.1667, A 0.000, B 0.000, C 0.000 }
gfCNCPoint1[22412] = {X 281.1776, Y 9.4435, Z -2.1667, A 0.000, B 0.000, C 0.000 }
gfCNCPoint1[22413] = {X 281.8743, Y 8.7468, Z -2.1667, A 0.000, B 0.000, C 0.000 }
gfCNCPoint1[22414] = {X 282.7086, Y 8.2226, Z -2.1667, A 0.000, B 0.000, C 0.000 }
gfCNCPoint1[22415] = {X 283.6386, Y 7.8971, Z -2.1667, A 0.000, B 0.000, C 0.000 }
gfCNCPoint1[22416] = {X 284.6177, Y 7.7868, Z -2.1667, A 0.000, B 0.000, C 0.000 }
gfCNCPoint1[22417] = {X 291.0611, Y 7.7868, Z -2.1667, A 0.000, B 0.000, C 0.000 }
gfCNCPoint1[22418] = {X 292.0402, Y 7.8971, Z -2.1667, A 0.000, B 0.000, C 0.000 }
gfCNCPoint1[22419] = {X 292.9702, Y 8.2226, Z -2.1667, A 0.000, B 0.000, C 0.000 }
gfCNCPoint1[22420] = {X 293.8045, Y 8.7468, Z -2.1667, A 0.000, B 0.000, C 0.000 }
gfCNCPoint1[22421] = {X 294.5012, Y 9.4435, Z -2.1667, A 0.000, B 0.000, C 0.000 }
gfCNCPoint1[22422] = {X 295.0254, Y 10.2777, Z -2.1667, A 0.000, B 0.000, C 0.000 }
gfCNCPoint1[22423] = {X 295.3508, Y 11.2077, Z -2.1667, A 0.000, B 0.000, C 0.000 }
gfCNCPoint1[22424] = {X 295.4611, Y 12.1868, Z -2.1667, A 0.000, B 0.000, C 0.000 }
gfCNCPoint1[22425] = {X 295.4609, Y 13.0233, Z -2.1667, A 0.000, B 0.000, C 0.000 }
gfCNCPoint1[22426] = {X 295.3525, Y 13.9496, Z -2.1667, A 0.000, B 0.000, C 0.000 }
gfCNCPoint1[22427] = {X 295.0513, Y 14.8323, Z -2.1667, A 0.000, B 0.000, C 0.000 }
gfCNCPoint1[22428] = {X 294.5708, Y 15.6317, Z -2.1667, A 0.000, B 0.000, C 0.000 }
gfCNCPoint1[22429] = {X 293.9327, Y 16.3118, Z -2.1667, A 0.000, B 0.000, C 0.000 }
gfCNCPoint1[22430] = {X 293.9340, Y 22.1165, Z -2.1667, A 0.000, B 0.000, C 0.000 }
gfCNCPoint1[22431] = {X 302.6797, Y 22.1165, Z -2.1667, A 0.000, B 0.000, C 0.000 }
gfCNCPoint1[22432] = {X 302.6803, Y 16.3115, Z -2.1667, A 0.000, B 0.000, C 0.000 }
gfCNCPoint1[22433] = {X 302.0355, Y 15.6223, Z -2.1667, A 0.000, B 0.000, C 0.000 }
gfCNCPoint1[22434] = {X 301.5524, Y 14.8115, Z -2.1667, A 0.000, B 0.000, C 0.000 }
gfCNCPoint1[22435] = {X 301.2535, Y 13.9163, Z -2.1667, A 0.000, B 0.000, C 0.000 }
gfCNCPoint1[22436] = {X 301.1523, Y 12.9779, Z -2.1667, A 0.000, B 0.000, C 0.000 }
gfCNCPoint1[22437] = {X 301.1523, Y 12.1868, Z -2.1667, A 0.000, B 0.000, C 0.000 }
gfCNCPoint1[22438] = {X 301.2626, Y 11.2077, Z -2.1667, A 0.000, B 0.000, C 0.000 }
gfCNCPoint1[22439] = {X 301.5880, Y 10.2777, Z -2.1667, A 0.000, B 0.000, C 0.000 }
gfCNCPoint1[22440] = {X 302.1122, Y 9.4435, Z -2.1667, A 0.000, B 0.000, C 0.000 }
gfCNCPoint1[22441] = {X 302.8089, Y 8.7468, Z -2.1667, A 0.000, B 0.000, C 0.000 }
gfCNCPoint1[22442] = {X 303.6432, Y 8.2226, Z -2.1667, A 0.000, B 0.000, C 0.000 }
gfCNCPoint1[22443] = {X 304.5732, Y 7.8971, Z -2.1667, A 0.000, B 0.000, C 0.000 }
gfCNCPoint1[22444] = {X 305.5523, Y 7.7868, Z -2.1667, A 0.000, B 0.000, C 0.000 }
gfCNCPoint1[22445] = {X 311.9957, Y 7.7868, Z -2.1667, A 0.000, B 0.000, C 0.000 }
gfCNCPoint1[22446] = {X 312.9748, Y 7.8971, Z -2.1667, A 0.000, B 0.000, C 0.000 }
gfCNCPoint1[22447] = {X 313.9048, Y 8.2226, Z -2.1667, A 0.000, B 0.000, C 0.000 }
gfCNCPoint1[22448] = {X 314.7391, Y 8.7468, Z -2.1667, A 0.000, B 0.000, C 0.000 }
gfCNCPoint1[22449] = {X 315.4358, Y 9.4435, Z -2.1667, A 0.000, B 0.000, C 0.000 }
gfCNCPoint1[22450] = {X 315.9600, Y 10.2777, Z -2.1667, A 0.000, B 0.000, C 0.000 }
gfCNCPoint1[22451] = {X 316.2854, Y 11.2077, Z -2.1667, A 0.000, B 0.000, C 0.000 }
gfCNCPoint1[22452] = {X 316.3957, Y 12.1868, Z -2.1667, A 0.000, B 0.000, C 0.000 }
gfCNCPoint1[22453] = {X 316.3955, Y 13.0233, Z -2.1667, A 0.000, B 0.000, C 0.000 }
gfCNCPoint1[22454] = {X 316.2871, Y 13.9496, Z -2.1667, A 0.000, B 0.000, C 0.000 }
gfCNCPoint1[22455] = {X 315.9860, Y 14.8322, Z -2.1667, A 0.000, B 0.000, C 0.000 }
gfCNCPoint1[22456] = {X 315.5055, Y 15.6315, Z -2.1667, A 0.000, B 0.000, C 0.000 }
gfCNCPoint1[22457] = {X 314.8674, Y 16.3117, Z -2.1667, A 0.000, B 0.000, C 0.000 }
gfCNCPoint1[22458] = {X 314.8672, Y 40.8749, Z -2.1667, A 0.000, B 0.000, C 0.000 }
gfCNCPoint1[22459] = {X 315.5122, Y 41.5641, Z -2.1667, A 0.000, B 0.000, C 0.000 }
gfCNCPoint1[22460] = {X 315.9954, Y 42.3751, Z -2.1667, A 0.000, B 0.000, C 0.000 }
gfCNCPoint1[22461] = {X 316.2945, Y 43.2704, Z -2.1667, A 0.000, B 0.000, C 0.000 }
gfCNCPoint1[22462] = {X 316.3957, Y 44.2089, Z -2.1667, A 0.000, B 0.000, C 0.000 }
gfCNCPoint1[22463] = {X 316.3957, Y 45.0000, Z -2.1667, A 0.000, B 0.000, C 0.000 }
gfCNCPoint1[22464] = {X 316.3190, Y 45.8182, Z -2.1667, A 0.000, B 0.000, C 0.000 }
gfCNCPoint1[22465] = {X 316.0914, Y 46.6079, Z -2.1667, A 0.000, B 0.000, C 0.000 }
gfCNCPoint1[22466] = {X 315.7209, Y 47.3415, Z -2.1667, A 0.000, B 0.000, C 0.000 }
gfCNCPoint1[22467] = {X 315.2205, Y 47.9934, Z -2.1667, A 0.000, B 0.000, C 0.000 }
gfCNCPoint1[22468] = {X 315.5723, Y 48.3200, Z -2.1667, A 0.000, B 0.000, C 0.000 }
gfCNCPoint1[22469] = {X 324.3107, Y 48.3200, Z -2.1667, A 0.000, B 0.000, C 0.000 }
gfCNCPoint1[22470] = {X 325.5555, Y 48.4004, Z -2.1667, A 0.000, B 0.000, C 0.000 }
gfCNCPoint1[22471] = {X 326.7797, Y 48.6402, Z -2.1667, A 0.000, B 0.000, C 0.000 }
gfCNCPoint1[22472] = {X 325.5882, Y 48.0963, Z -2.1667, A 0.000, B 0.000, C 0.000 }
gfCNCPoint1[22473] = {X 324.4810, Y 47.3966, Z -2.1667, A 0.000, B 0.000, C 0.000 }
gfCNCPoint1[22474] = {X 323.4784, Y 46.5538, Z -2.1667, A 0.000, B 0.000, C 0.000 }
gfCNCPoint1[22475] = {X 322.8382, Y 45.9295, Z -2.1667, A 0.000, B 0.000, C 0.000 }
gfCNCPoint1[22476] = {X 322.2180, Y 45.2650, Z -2.1667, A 0.000, B 0.000, C 0.000 }
gfCNCPoint1[22477] = {X 321.6628, Y 44.5452, Z -2.1667, A 0.000, B 0.000, C 0.000 }
gfCNCPoint1[22478] = {X 323.6300, Y 43.1703, Z -2.1667, A 0.000, B 0.000, C 0.000 }
gfCNCPoint1[22479] = {X 323.0063, Y 42.0918, Z -2.1667, A 0.000, B 0.000, C 0.000 }
gfCNCPoint1[22480] = {X 322.5757, Y 40.9227, Z -2.1667, A 0.000, B 0.000, C 0.000 }
gfCNCPoint1[22481] = {X 322.3506, Y 39.6973, Z -2.1667, A 0.000, B 0.000, C 0.000 }
gfCNCPoint1[22482] = {X 322.3379, Y 38.4514, Z -2.1667, A 0.000, B 0.000, C 0.000 }
gfCNCPoint1[22483] = {X 322.5377, Y 37.2217, Z -2.1667, A 0.000, B 0.000, C 0.000 }
gfCNCPoint1[22484] = {X 322.9443, Y 36.0440, Z -2.1667, A 0.000, B 0.000, C 0.000 }
gfCNCPoint1[22485] = {X 323.5458, Y 34.9529, Z -2.1667, A 0.000, B 0.000, C 0.000 }
gfCNCPoint1[22486] = {X 327.7841, Y 28.6157, Z -2.1667, A 0.000, B 0.000, C 0.000 }
gfCNCPoint1[22487] = {X 328.5200, Y 27.6906, Z -2.1667, A 0.000, B 0.000, C 0.000 }
gfCNCPoint1[22488] = {X 329.3960, Y 26.8968, Z -2.1667, A 0.000, B 0.000, C 0.000 }
gfCNCPoint1[22489] = {X 330.3889, Y 26.2552, Z -2.1667, A 0.000, B 0.000, C 0.000 }
gfCNCPoint1[22490] = {X 331.5063, Y 25.7713, Z -2.1667, A 0.000, B 0.000, C 0.000 }
gfCNCPoint1[22491] = {X 332.6887, Y 25.4804, Z -2.1667, A 0.000, B 0.000, C 0.000 }
gfCNCPoint1[22492] = {X 333.9031, Y 25.3907, Z -2.1667, A 0.000, B 0.000, C 0.000 }
gfCNCPoint1[22493] = {X 335.1154, Y 25.5046, Z -2.1667, A 0.000, B 0.000, C 0.000 }
gfCNCPoint1[22494] = {X 336.2918, Y 25.8191, Z -2.1667, A 0.000, B 0.000, C 0.000 }
gfCNCPoint1[22495] = {X 337.3993, Y 26.3252, Z -2.1667, A 0.000, B 0.000, C 0.000 }
gfCNCPoint1[22496] = {X 338.1754, Y 26.8291, Z -2.1667, A 0.000, B 0.000, C 0.000 }
gfCNCPoint1[22497] = {X 338.8813, Y 27.4275, Z -2.1667, A 0.000, B 0.000, C 0.000 }
gfCNCPoint1[22498] = {X 339.4514, Y 27.9767, Z -2.1667, A 0.000, B 0.000, C 0.000 }
gfCNCPoint1[22499] = {X 339.8232, Y 28.3622, Z -2.1667, A 0.000, B 0.000, C 0.000 }
gfCNCPoint1[22500] = {X 340.1656, Y 28.7740, Z -2.1667, A 0.000, B 0.000, C 0.000 }
gfCNCPoint1[22501] = {X 345.8671, Y 24.3770, Z -2.1667, A 0.000, B 0.000, C 0.000 }
gfCNCPoint1[22502] = {X 346.4662, Y 25.2138, Z -2.1667, A 0.000, B 0.000, C 0.000 }
gfCNCPoint1[22503] = {X 347.0044, Y 26.0909, Z -2.1667, A 0.000, B 0.000, C 0.000 }
gfCNCPoint1[22504] = {X 347.1184, Y 24.7348, Z -2.1667, A 0.000, B 0.000, C 0.000 }
gfCNCPoint1[22505] = {X 346.9945, Y 23.3795, Z -2.1667, A 0.000, B 0.000, C 0.000 }
gfCNCPoint1[22506] = {X 346.9504, Y 23.1695, Z -2.1667, A 0.000, B 0.000, C 0.000 }
gfCNCPoint1[22507] = {X 346.8822, Y 22.9661, Z -2.1667, A 0.000, B 0.000, C 0.000 }
gfCNCPoint1[22508] = {X 346.3958, Y 23.6868, Z -2.1667, A 0.000, B 0.000, C 0.000 }
gfCNCPoint1[22509] = {X 345.8671, Y 24.3770, Z -2.1667, A 0.000, B 0.000, C 0.000 }
gfCNCPoint1[22510] = {X 343.9666, Y 25.8427, Z -2.1667, A 0.000, B 0.000, C 0.000 }
gfCNCPoint1[22511] = {X 344.4664, Y 26.5407, Z -2.1667, A 0.000, B 0.000, C 0.000 }
gfCNCPoint1[22512] = {X 344.9154, Y 27.2725, Z -2.1667, A 0.000, B 0.000, C 0.000 }
gfCNCPoint1[22513] = {X 345.4671, Y 28.3758, Z -2.1667, A 0.000, B 0.000, C 0.000 }
gfCNCPoint1[22514] = {X 345.9034, Y 29.5297, Z -2.1667, A 0.000, B 0.000, C 0.000 }
gfCNCPoint1[22515] = {X 346.4600, Y 29.6323, Z -2.1667, A 0.000, B 0.000, C 0.000 }
gfCNCPoint1[22516] = {X 347.0259, Y 29.6231, Z -2.1667, A 0.000, B 0.000, C 0.000 }
gfCNCPoint1[22517] = {X 347.4365, Y 29.5576, Z -2.1667, A 0.000, B 0.000, C 0.000 }
gfCNCPoint1[22518] = {X 347.7959, Y 29.3488, Z -2.1667, A 0.000, B 0.000, C 0.000 }
gfCNCPoint1[22519] = {X 348.4758, Y 28.6282, Z -2.1667, A 0.000, B 0.000, C 0.000 }
gfCNCPoint1[22520] = {X 348.9864, Y 27.7792, Z -2.1667, A 0.000, B 0.000, C 0.000 }
gfCNCPoint1[22521] = {X 349.3042, Y 26.8409, Z -2.1667, A 0.000, B 0.000, C 0.000 }
gfCNCPoint1[22522] = {X 349.3381, Y 26.6709, Z -2.1667, A 0.000, B 0.000, C 0.000 }
gfCNCPoint1[22523] = {X 349.3692, Y 26.5004, Z -2.1667, A 0.000, B 0.000, C 0.000 }
gfCNCPoint1[22524] = {X 349.5028, Y 25.3288, Z -2.1667, A 0.000, B 0.000, C 0.000 }
gfCNCPoint1[22525] = {X 349.5000, Y 24.1496, Z -2.1667, A 0.000, B 0.000, C 0.000 }
gfCNCPoint1[22526] = {X 349.3609, Y 22.9786, Z -2.1667, A 0.000, B 0.000, C 0.000 }
gfCNCPoint1[22527] = {X 349.1890, Y 22.2868, Z -2.1667, A 0.000, B 0.000, C 0.000 }
gfCNCPoint1[22528] = {X 348.9036, Y 21.6335, Z -2.1667, A 0.000, B 0.000, C 0.000 }
gfCNCPoint1[22529] = {X 348.5128, Y 21.0373, Z -2.1667, A 0.000, B 0.000, C 0.000 }
gfCNCPoint1[22530] = {X 348.1202, Y 20.6779, Z -2.1667, A 0.000, B 0.000, C 0.000 }
gfCNCPoint1[22531] = {X 347.6258, Y 20.4807, Z -2.1667, A 0.000, B 0.000, C 0.000 }
gfCNCPoint1[22532] = {X 346.5729, Y 20.3822, Z -2.1667, A 0.000, B 0.000, C 0.000 }
gfCNCPoint1[22533] = {X 345.5201, Y 20.4825, Z -2.1667, A 0.000, B 0.000, C 0.000 }
gfCNCPoint1[22534] = {X 344.7179, Y 21.8934, Z -2.1667, A 0.000, B 0.000, C 0.000 }
gfCNCPoint1[22535] = {X 343.7339, Y 23.1840, Z -2.1667, A 0.000, B 0.000, C 0.000 }
gfCNCPoint1[22536] = {X 342.5857, Y 24.3311, Z -2.1667, A 0.000, B 0.000, C 0.000 }
gfCNCPoint1[22537] = {X 342.7814, Y 24.5197, Z -2.1667, A 0.000, B 0.000, C 0.000 }
gfCNCPoint1[22538] = {X 343.3984, Y 25.1594, Z -2.1667, A 0.000, B 0.000, C 0.000 }
gfCNCPoint1[22539] = {X 343.9666, Y 25.8427, Z -2.1667, A 0.000, B 0.000, C 0.000 }
gfCNCPoint1[22540] = {X 342.0661, Y 27.3083, Z -2.1667, A 0.000, B 0.000, C 0.000 }
gfCNCPoint1[22541] = {X 342.8615, Y 28.5166, Z -2.1667, A 0.000, B 0.000, C 0.000 }
gfCNCPoint1[22542] = {X 343.4678, Y 29.8299, Z -2.1667, A 0.000, B 0.000, C 0.000 }
gfCNCPoint1[22543] = {X 343.8718, Y 31.2189, Z -2.1667, A 0.000, B 0.000, C 0.000 }
gfCNCPoint1[22544] = {X 344.6368, Y 31.6218, Z -2.1667, A 0.000, B 0.000, C 0.000 }
gfCNCPoint1[22545] = {X 345.4576, Y 31.8938, Z -2.1667, A 0.000, B 0.000, C 0.000 }
gfCNCPoint1[22546] = {X 346.3118, Y 32.0276, Z -2.1667, A 0.000, B 0.000, C 0.000 }
gfCNCPoint1[22547] = {X 347.1765, Y 32.0194, Z -2.1667, A 0.000, B 0.000, C 0.000 }
gfCNCPoint1[22548] = {X 347.9605, Y 31.9042, Z -2.1667, A 0.000, B 0.000, C 0.000 }
gfCNCPoint1[22549] = {X 348.6992, Y 31.6173, Z -2.1667, A 0.000, B 0.000, C 0.000 }
gfCNCPoint1[22550] = {X 349.3554, Y 31.1731, Z -2.1667, A 0.000, B 0.000, C 0.000 }
gfCNCPoint1[22551] = {X 350.1553, Y 30.3690, Z -2.1667, A 0.000, B 0.000, C 0.000 }
gfCNCPoint1[22552] = {X 350.8152, Y 29.4467, Z -2.1667, A 0.000, B 0.000, C 0.000 }
gfCNCPoint1[22553] = {X 351.3180, Y 28.4302, Z -2.1667, A 0.000, B 0.000, C 0.000 }
gfCNCPoint1[22554] = {X 351.6505, Y 27.3459, Z -2.1667, A 0.000, B 0.000, C 0.000 }
gfCNCPoint1[22555] = {X 351.8787, Y 25.7633, Z -2.1667, A 0.000, B 0.000, C 0.000 }
gfCNCPoint1[22556] = {X 351.9042, Y 24.1645, Z -2.1667, A 0.000, B 0.000, C 0.000 }
gfCNCPoint1[22557] = {X 351.7268, Y 22.5754, Z -2.1667, A 0.000, B 0.000, C 0.000 }
gfCNCPoint1[22558] = {X 351.4579, Y 21.5045, Z -2.1667, A 0.000, B 0.000, C 0.000 }
gfCNCPoint1[22559] = {X 351.0152, Y 20.4929, Z -2.1667, A 0.000, B 0.000, C 0.000 }
gfCNCPoint1[22560] = {X 350.4110, Y 19.5687, Z -2.1667, A 0.000, B 0.000, C 0.000 }
gfCNCPoint1[22561] = {X 349.7599, Y 18.9039, Z -2.1667, A 0.000, B 0.000, C 0.000 }
gfCNCPoint1[22562] = {X 348.9693, Y 18.4132, Z -2.1667, A 0.000, B 0.000, C 0.000 }
gfCNCPoint1[22563] = {X 348.0846, Y 18.1249, Z -2.1667, A 0.000, B 0.000, C 0.000 }
gfCNCPoint1[22564] = {X 346.9931, Y 17.9929, Z -2.1667, A 0.000, B 0.000, C 0.000 }
gfCNCPoint1[22565] = {X 345.8939, Y 18.0114, Z -2.1667, A 0.000, B 0.000, C 0.000 }
gfCNCPoint1[22566] = {X 344.8075, Y 18.1799, Z -2.1667, A 0.000, B 0.000, C 0.000 }
gfCNCPoint1[22567] = {X 343.7543, Y 18.4953, Z -2.1667, A 0.000, B 0.000, C 0.000 }
gfCNCPoint1[22568] = {X 343.2662, Y 19.6257, Z -2.1667, A 0.000, B 0.000, C 0.000 }
gfCNCPoint1[22569] = {X 342.6386, Y 20.6850, Z -2.1667, A 0.000, B 0.000, C 0.000 }
gfCNCPoint1[22570] = {X 341.8815, Y 21.6560, Z -2.1667, A 0.000, B 0.000, C 0.000 }
gfCNCPoint1[22571] = {X 341.0073, Y 22.5231, Z -2.1667, A 0.000, B 0.000, C 0.000 }
gfCNCPoint1[22572] = {X 340.7217, Y 22.7629, Z -2.1667, A 0.000, B 0.000, C 0.000 }
gfCNCPoint1[22573] = {X 340.4270, Y 22.9916, Z -2.1667, A 0.000, B 0.000, C 0.000 }
gfCNCPoint1[22574] = {X 339.6615, Y 23.5549, Z -2.1667, A 0.000, B 0.000, C 0.000 }
gfCNCPoint1[22575] = {X 339.1299, Y 23.9121, Z -2.1667, A 0.000, B 0.000, C 0.000 }
gfCNCPoint1[22576] = {X 338.5759, Y 24.2333, Z -2.1667, A 0.000, B 0.000, C 0.000 }
gfCNCPoint1[22577] = {X 339.6078, Y 24.9035, Z -2.1667, A 0.000, B 0.000, C 0.000 }
gfCNCPoint1[22578] = {X 340.5464, Y 25.6991, Z -2.1667, A 0.000, B 0.000, C 0.000 }
gfCNCPoint1[22579] = {X 341.1164, Y 26.2482, Z -2.1667, A 0.000, B 0.000, C 0.000 }
gfCNCPoint1[22580] = {X 341.6108, Y 26.7608, Z -2.1667, A 0.000, B 0.000, C 0.000 }
gfCNCPoint1[22581] = {X 342.0661, Y 27.3083, Z -2.1667, A 0.000, B 0.000, C 0.000 }
gfCNCPoint1[22582] = {X 340.1656, Y 28.7740, Z -2.1667, A 0.000, B 0.000, C 0.000 }
gfCNCPoint1[22583] = {X 340.7342, Y 29.6299, Z -2.1667, A 0.000, B 0.000, C 0.000 }
gfCNCPoint1[22584] = {X 341.1765, Y 30.5574, Z -2.1667, A 0.000, B 0.000, C 0.000 }
gfCNCPoint1[22585] = {X 341.4839, Y 31.5378, Z -2.1667, A 0.000, B 0.000, C 0.000 }
gfCNCPoint1[22586] = {X 341.6501, Y 32.5518, Z -2.1667, A 0.000, B 0.000, C 0.000 }
gfCNCPoint1[22587] = {X 341.8441, Y 32.7094, Z -2.1667, A 0.000, B 0.000, C 0.000 }
gfCNCPoint1[22588] = {X 342.0404, Y 32.8641, Z -2.1667, A 0.000, B 0.000, C 0.000 }
gfCNCPoint1[22589] = {X 342.9833, Y 33.4816, Z -2.1667, A 0.000, B 0.000, C 0.000 }
gfCNCPoint1[22590] = {X 344.0067, Y 33.9540, Z -2.1667, A 0.000, B 0.000, C 0.000 }
gfCNCPoint1[22591] = {X 345.0883, Y 34.2710, Z -2.1667, A 0.000, B 0.000, C 0.000 }
gfCNCPoint1[22592] = {X 346.2048, Y 34.4257, Z -2.1667, A 0.000, B 0.000, C 0.000 }
gfCNCPoint1[22593] = {X 347.3318, Y 34.4148, Z -2.1667, A 0.000, B 0.000, C 0.000 }
gfCNCPoint1[22594] = {X 348.3036, Y 34.2889, Z -2.1667, A 0.000, B 0.000, C 0.000 }
gfCNCPoint1[22595] = {X 349.2414, Y 34.0049, Z -2.1667, A 0.000, B 0.000, C 0.000 }
gfCNCPoint1[22596] = {X 350.1198, Y 33.5705, Z -2.1667, A 0.000, B 0.000, C 0.000 }
gfCNCPoint1[22597] = {X 350.9147, Y 32.9975, Z -2.1667, A 0.000, B 0.000, C 0.000 }
gfCNCPoint1[22598] = {X 351.7891, Y 32.1463, Z -2.1667, A 0.000, B 0.000, C 0.000 }
gfCNCPoint1[22599] = {X 352.5462, Y 31.1891, Z -2.1667, A 0.000, B 0.000, C 0.000 }
gfCNCPoint1[22600] = {X 353.1731, Y 30.1420, Z -2.1667, A 0.000, B 0.000, C 0.000 }
gfCNCPoint1[22601] = {X 353.6595, Y 29.0227, Z -2.1667, A 0.000, B 0.000, C 0.000 }
gfCNCPoint1[22602] = {X 353.9970, Y 27.8500, Z -2.1667, A 0.000, B 0.000, C 0.000 }
gfCNCPoint1[22603] = {X 354.2243, Y 26.4402, Z -2.1667, A 0.000, B 0.000, C 0.000 }
gfCNCPoint1[22604] = {X 354.3164, Y 25.0152, Z -2.1667, A 0.000, B 0.000, C 0.000 }
gfCNCPoint1[22605] = {X 354.2723, Y 23.5879, Z -2.1667, A 0.000, B 0.000, C 0.000 }
gfCNCPoint1[22606] = {X 354.0926, Y 22.1713, Z -2.1667, A 0.000, B 0.000, C 0.000 }
gfCNCPoint1[22607] = {X 353.8399, Y 21.0759, Z -2.1667, A 0.000, B 0.000, C 0.000 }
gfCNCPoint1[22608] = {X 353.4532, Y 20.0203, Z -2.1667, A 0.000, B 0.000, C 0.000 }
gfCNCPoint1[22609] = {X 352.9385, Y 19.0209, Z -2.1667, A 0.000, B 0.000, C 0.000 }
gfCNCPoint1[22610] = {X 352.3038, Y 18.0931, Z -2.1667, A 0.000, B 0.000, C 0.000 }
gfCNCPoint1[22611] = {X 351.5368, Y 17.2657, Z -2.1667, A 0.000, B 0.000, C 0.000 }
gfCNCPoint1[22612] = {X 350.6342, Y 16.5889, Z -2.1667, A 0.000, B 0.000, C 0.000 }
gfCNCPoint1[22613] = {X 349.6250, Y 16.0845, Z -2.1667, A 0.000, B 0.000, C 0.000 }
gfCNCPoint1[22614] = {X 348.5419, Y 15.7689, Z -2.1667, A 0.000, B 0.000, C 0.000 }
gfCNCPoint1[22615] = {X 347.1562, Y 15.5982, Z -2.1667, A 0.000, B 0.000, C 0.000 }
gfCNCPoint1[22616] = {X 345.7601, Y 15.6143, Z -2.1667, A 0.000, B 0.000, C 0.000 }
gfCNCPoint1[22617] = {X 344.3787, Y 15.8168, Z -2.1667, A 0.000, B 0.000, C 0.000 }
gfCNCPoint1[22618] = {X 343.0367, Y 16.2021, Z -2.1667, A 0.000, B 0.000, C 0.000 }
gfCNCPoint1[22619] = {X 341.7583, Y 16.7632, Z -2.1667, A 0.000, B 0.000, C 0.000 }
gfCNCPoint1[22620] = {X 341.3709, Y 18.0079, Z -2.1667, A 0.000, B 0.000, C 0.000 }
gfCNCPoint1[22621] = {X 340.7677, Y 19.1636, Z -2.1667, A 0.000, B 0.000, C 0.000 }
gfCNCPoint1[22622] = {X 339.9681, Y 20.1932, Z -2.1667, A 0.000, B 0.000, C 0.000 }
gfCNCPoint1[22623] = {X 338.9976, Y 21.0636, Z -2.1667, A 0.000, B 0.000, C 0.000 }
gfCNCPoint1[22624] = {X 338.2497, Y 21.6140, Z -2.1667, A 0.000, B 0.000, C 0.000 }
gfCNCPoint1[22625] = {X 337.8538, Y 21.8795, Z -2.1667, A 0.000, B 0.000, C 0.000 }
gfCNCPoint1[22626] = {X 337.4413, Y 22.1185, Z -2.1667, A 0.000, B 0.000, C 0.000 }
gfCNCPoint1[22627] = {X 336.3239, Y 22.6023, Z -2.1667, A 0.000, B 0.000, C 0.000 }
gfCNCPoint1[22628] = {X 335.1415, Y 22.8932, Z -2.1667, A 0.000, B 0.000, C 0.000 }
gfCNCPoint1[22629] = {X 333.9271, Y 22.9829, Z -2.1667, A 0.000, B 0.000, C 0.000 }
gfCNCPoint1[22630] = {X 332.7148, Y 22.8690, Z -2.1667, A 0.000, B 0.000, C 0.000 }
gfCNCPoint1[22631] = {X 331.5384, Y 22.5546, Z -2.1667, A 0.000, B 0.000, C 0.000 }
gfCNCPoint1[22632] = {X 330.4309, Y 22.0485, Z -2.1667, A 0.000, B 0.000, C 0.000 }
gfCNCPoint1[22633] = {X 329.5143, Y 21.4374, Z -2.1667, A 0.000, B 0.000, C 0.000 }
gfCNCPoint1[22634] = {X 328.7005, Y 20.6950, Z -2.1667, A 0.000, B 0.000, C 0.000 }
gfCNCPoint1[22635] = {X 328.0080, Y 19.8382, Z -2.1667, A 0.000, B 0.000, C 0.000 }
gfCNCPoint1[22636] = {X 327.4528, Y 18.8869, Z -2.1667, A 0.000, B 0.000, C 0.000 }
gfCNCPoint1[22637] = {X 323.9321, Y 11.6443, Z -2.1667, A 0.000, B 0.000, C 0.000 }
gfCNCPoint1[22638] = {X 323.5337, Y 10.6422, Z -2.1667, A 0.000, B 0.000, C 0.000 }
gfCNCPoint1[22639] = {X 323.2878, Y 9.5922, Z -2.1667, A 0.000, B 0.000, C 0.000 }
gfCNCPoint1[22640] = {X 323.1997, Y 8.5174, Z -2.1667, A 0.000, B 0.000, C 0.000 }
gfCNCPoint1[22641] = {X 323.2713, Y 7.4414, Z -2.1667, A 0.000, B 0.000, C 0.000 }
gfCNCPoint1[22642] = {X 323.4719, Y 6.4885, Z -2.1667, A 0.000, B 0.000, C 0.000 }
gfCNCPoint1[22643] = {X 323.7979, Y 5.5709, Z -2.1667, A 0.000, B 0.000, C 0.000 }
gfCNCPoint1[22644] = {X 324.2435, Y 4.7051, Z -2.1667, A 0.000, B 0.000, C 0.000 }
gfCNCPoint1[22645] = {X 168.0205, Y 4.7051, Z -2.1667, A 0.000, B 0.000, C 0.000 }
gfCNCPoint1[22646] = {X 168.0205, Y 9.5051, Z -2.1667, A 0.000, B 0.000, C 0.000 }
gfCNCPoint1[22647] = {X 166.5360, Y 9.5051, Z -2.1667, A 0.000, B 0.000, C 0.000 }
gfCNCPoint1[22648] = {X 166.5856, Y 9.9932, Z -2.1667, A 0.000, B 0.000, C 0.000 }
gfCNCPoint1[22649] = {X 166.6021, Y 10.4835, Z -2.1667, A 0.000, B 0.000, C 0.000 }
gfCNCPoint1[22650] = {X 166.6021, Y 13.0969, Z -2.1667, A 0.000, B 0.000, C 0.000 }
gfCNCPoint1[22651] = {X 166.8569, Y 11.8210, Z -2.1667, A 0.000, B 0.000, C 0.000 }
gfCNCPoint1[22652] = {X 167.3348, Y 10.6108, Z -2.1667, A 0.000, B 0.000, C 0.000 }
gfCNCPoint1[22653] = {X 168.0205, Y 9.5051, Z -2.1667, A 0.000, B 0.000, C 0.000 }
gfCNCPoint1[22654] = {X 168.0205, Y 7.1051, Z -2.1667, A 0.000, B 0.000, C 0.000 }
gfCNCPoint1[22655] = {X 162.8435, Y 7.1051, Z -2.1667, A 0.000, B 0.000, C 0.000 }
gfCNCPoint1[22656] = {X 163.4703, Y 7.9132, Z -2.1667, A 0.000, B 0.000, C 0.000 }
gfCNCPoint1[22657] = {X 163.9149, Y 8.8342, Z -2.1667, A 0.000, B 0.000, C 0.000 }
gfCNCPoint1[22658] = {X 164.1578, Y 9.8276, Z -2.1667, A 0.000, B 0.000, C 0.000 }
gfCNCPoint1[22659] = {X 164.1910, Y 10.1548, Z -2.1667, A 0.000, B 0.000, C 0.000 }
gfCNCPoint1[22660] = {X 164.2021, Y 10.4835, Z -2.1667, A 0.000, B 0.000, C 0.000 }
gfCNCPoint1[22661] = {X 164.2021, Y 17.4615, Z -2.1667, A 0.000, B 0.000, C 0.000 }
gfCNCPoint1[22662] = {X 164.1140, Y 18.3848, Z -2.1667, A 0.000, B 0.000, C 0.000 }
gfCNCPoint1[22663] = {X 163.8527, Y 19.2747, Z -2.1667, A 0.000, B 0.000, C 0.000 }
gfCNCPoint1[22664] = {X 163.4279, Y 20.0991, Z -2.1667, A 0.000, B 0.000, C 0.000 }
gfCNCPoint1[22665] = {X 162.8547, Y 20.8283, Z -2.1667, A 0.000, B 0.000, C 0.000 }
gfCNCPoint1[22666] = {X 162.1540, Y 21.4358, Z -2.1667, A 0.000, B 0.000, C 0.000 }
gfCNCPoint1[22667] = {X 161.3509, Y 21.8998, Z -2.1667, A 0.000, B 0.000, C 0.000 }
gfCNCPoint1[22668] = {X 160.4746, Y 22.2035, Z -2.1667, A 0.000, B 0.000, C 0.000 }
gfCNCPoint1[22669] = {X 162.1750, Y 29.1998, Z -2.1667, A 0.000, B 0.000, C 0.000 }
gfCNCPoint1[22670] = {X 161.1122, Y 29.4082, Z -2.1667, A 0.000, B 0.000, C 0.000 }
gfCNCPoint1[22671] = {X 160.0350, Y 29.5205, Z -2.1667, A 0.000, B 0.000, C 0.000 }
gfCNCPoint1[22672] = {X 160.0343, Y 38.3366, Z -2.1667, A 0.000, B 0.000, C 0.000 }
gfCNCPoint1[22673] = {X 160.6825, Y 39.6937, Z -2.1667, A 0.000, B 0.000, C 0.000 }
gfCNCPoint1[22674] = {X 161.1577, Y 41.1206, Z -2.1667, A 0.000, B 0.000, C 0.000 }
gfCNCPoint1[22675] = {X 162.0487, Y 41.1205, Z -2.1667, A 0.000, B 0.000, C 0.000 }
gfCNCPoint1[22676] = {X 161.6745, Y 39.3711, Z -2.1667, A 0.000, B 0.000, C 0.000 }
gfCNCPoint1[22677] = {X 161.4505, Y 37.5962, Z -2.1667, A 0.000, B 0.000, C 0.000 }
gfCNCPoint1[22678] = {X 161.3321, Y 35.4807, Z -2.1667, A 0.000, B 0.000, C 0.000 }
gfCNCPoint1[22679] = {X 161.4142, Y 33.3636, Z -2.1667, A 0.000, B 0.000, C 0.000 }
gfCNCPoint1[22680] = {X 161.6960, Y 31.2637, Z -2.1667, A 0.000, B 0.000, C 0.000 }
gfCNCPoint1[22681] = {X 162.1750, Y 29.1998, Z -2.1667, A 0.000, B 0.000, C 0.000 }
gfCNCPoint1[22682] = {X 161.6082, Y 26.8677, Z -2.1667, A 0.000, B 0.000, C 0.000 }
gfCNCPoint1[22683] = {X 160.4733, Y 27.0728, Z -2.1667, A 0.000, B 0.000, C 0.000 }
gfCNCPoint1[22684] = {X 159.3220, Y 27.1415, Z -2.1667, A 0.000, B 0.000, C 0.000 }
gfCNCPoint1[22685] = {X 158.6676, Y 27.1415, Z -2.1667, A 0.000, B 0.000, C 0.000 }
gfCNCPoint1[22686] = {X 158.1506, Y 27.1260, Z -2.1667, A 0.000, B 0.000, C 0.000 }
gfCNCPoint1[22687] = {X 157.6352, Y 27.0830, Z -2.1667, A 0.000, B 0.000, C 0.000 }
gfCNCPoint1[22688] = {X 157.6343, Y 38.9961, Z -2.1667, A 0.000, B 0.000, C 0.000 }
gfCNCPoint1[22689] = {X 158.2181, Y 40.0485, Z -2.1667, A 0.000, B 0.000, C 0.000 }
gfCNCPoint1[22690] = {X 158.6675, Y 41.1649, Z -2.1667, A 0.000, B 0.000, C 0.000 }
gfCNCPoint1[22691] = {X 158.9754, Y 42.3283, Z -2.1667, A 0.000, B 0.000, C 0.000 }
gfCNCPoint1[22692] = {X 159.1373, Y 43.5209, Z -2.1667, A 0.000, B 0.000, C 0.000 }
gfCNCPoint1[22693] = {X 165.4305, Y 43.5200, Z -2.1667, A 0.000, B 0.000, C 0.000 }
gfCNCPoint1[22694] = {X 164.8370, Y 42.0421, Z -2.1667, A 0.000, B 0.000, C 0.000 }
gfCNCPoint1[22695] = {X 164.3721, Y 40.5189, Z -2.1667, A 0.000, B 0.000, C 0.000 }
gfCNCPoint1[22696] = {X 164.0386, Y 38.9574, Z -2.1667, A 0.000, B 0.000, C 0.000 }
gfCNCPoint1[22697] = {X 163.8402, Y 37.3732, Z -2.1667, A 0.000, B 0.000, C 0.000 }
gfCNCPoint1[22698] = {X 163.7322, Y 35.4785, Z -2.1667, A 0.000, B 0.000, C 0.000 }
gfCNCPoint1[22699] = {X 163.8042, Y 33.5821, Z -2.1667, A 0.000, B 0.000, C 0.000 }
gfCNCPoint1[22700] = {X 164.0558, Y 31.7011, Z -2.1667, A 0.000, B 0.000, C 0.000 }
gfCNCPoint1[22701] = {X 164.4846, Y 29.8524, Z -2.1667, A 0.000, B 0.000, C 0.000 }
gfCNCPoint1[22702] = {X 164.8365, Y 28.7334, Z -2.1667, A 0.000, B 0.000, C 0.000 }
gfCNCPoint1[22703] = {X 165.2535, Y 27.6370, Z -2.1667, A 0.000, B 0.000, C 0.000 }
gfCNCPoint1[22704] = {X 165.8702, Y 26.3063, Z -2.1667, A 0.000, B 0.000, C 0.000 }
gfCNCPoint1[22705] = {X 166.6045, Y 25.0366, Z -2.1667, A 0.000, B 0.000, C 0.000 }
gfCNCPoint1[22706] = {X 167.4505, Y 23.8385, Z -2.1667, A 0.000, B 0.000, C 0.000 }
gfCNCPoint1[22707] = {X 167.1640, Y 23.1367, Z -2.1667, A 0.000, B 0.000, C 0.000 }
gfCNCPoint1[22708] = {X 166.2874, Y 24.1837, Z -2.1667, A 0.000, B 0.000, C 0.000 }
gfCNCPoint1[22709] = {X 165.2721, Y 25.0969, Z -2.1667, A 0.000, B 0.000, C 0.000 }
gfCNCPoint1[22710] = {X 164.1385, Y 25.8582, Z -2.1667, A 0.000, B 0.000, C 0.000 }
gfCNCPoint1[22711] = {X 162.9090, Y 26.4524, Z -2.1667, A 0.000, B 0.000, C 0.000 }
gfCNCPoint1[22712] = {X 161.6082, Y 26.8677, Z -2.1667, A 0.000, B 0.000, C 0.000 }
gfCNCPoint1[22713] = {X 161.0414, Y 24.5356, Z -2.1667, A 0.000, B 0.000, C 0.000 }
gfCNCPoint1[22714] = {X 160.1878, Y 24.6899, Z -2.1667, A 0.000, B 0.000, C 0.000 }
gfCNCPoint1[22715] = {X 159.3220, Y 24.7415, Z -2.1667, A 0.000, B 0.000, C 0.000 }
gfCNCPoint1[22716] = {X 158.6757, Y 24.7415, Z -2.1667, A 0.000, B 0.000, C 0.000 }
gfCNCPoint1[22717] = {X 158.2864, Y 24.7299, Z -2.1667, A 0.000, B 0.000, C 0.000 }
gfCNCPoint1[22718] = {X 157.8982, Y 24.6975, Z -2.1667, A 0.000, B 0.000, C 0.000 }
gfCNCPoint1[22719] = {X 156.9777, Y 24.5359, Z -2.1667, A 0.000, B 0.000, C 0.000 }
gfCNCPoint1[22720] = {X 156.0852, Y 24.2584, Z -2.1667, A 0.000, B 0.000, C 0.000 }
gfCNCPoint1[22721] = {X 155.2354, Y 23.8694, Z -2.1667, A 0.000, B 0.000, C 0.000 }
gfCNCPoint1[22722] = {X 155.2342, Y 39.7517, Z -2.1667, A 0.000, B 0.000, C 0.000 }
gfCNCPoint1[22723] = {X 155.8250, Y 40.6439, Z -2.1667, A 0.000, B 0.000, C 0.000 }
gfCNCPoint1[22724] = {X 156.2795, Y 41.6126, Z -2.1667, A 0.000, B 0.000, C 0.000 }
gfCNCPoint1[22725] = {X 156.5879, Y 42.6372, Z -2.1667, A 0.000, B 0.000, C 0.000 }
gfCNCPoint1[22726] = {X 156.7437, Y 43.6958, Z -2.1667, A 0.000, B 0.000, C 0.000 }
gfCNCPoint1[22727] = {X 156.7578, Y 43.9498, Z -2.1667, A 0.000, B 0.000, C 0.000 }
gfCNCPoint1[22728] = {X 156.7631, Y 44.2042, Z -2.1667, A 0.000, B 0.000, C 0.000 }
gfCNCPoint1[22729] = {X 156.7629, Y 45.0588, Z -2.1667, A 0.000, B 0.000, C 0.000 }
gfCNCPoint1[22730] = {X 156.7352, Y 45.6370, Z -2.1667, A 0.000, B 0.000, C 0.000 }
gfCNCPoint1[22731] = {X 156.6616, Y 46.2112, Z -2.1667, A 0.000, B 0.000, C 0.000 }
gfCNCPoint1[22732] = {X 157.9052, Y 46.0006, Z -2.1667, A 0.000, B 0.000, C 0.000 }
gfCNCPoint1[22733] = {X 159.1639, Y 45.9207, Z -2.1667, A 0.000, B 0.000, C 0.000 }
gfCNCPoint1[22734] = {X 159.2309, Y 45.9202, Z -2.1667, A 0.000, B 0.000, C 0.000 }
gfCNCPoint1[22735] = {X 159.2980, Y 45.9200, Z -2.1667, A 0.000, B 0.000, C 0.000 }
gfCNCPoint1[22736] = {X 169.6839, Y 45.9200, Z -2.1667, A 0.000, B 0.000, C 0.000 }
gfCNCPoint1[22737] = {X 168.9032, Y 44.8481, Z -2.1667, A 0.000, B 0.000, C 0.000 }
gfCNCPoint1[22738] = {X 168.2128, Y 43.7159, Z -2.1667, A 0.000, B 0.000, C 0.000 }
gfCNCPoint1[22739] = {X 167.6173, Y 42.5310, Z -2.1667, A 0.000, B 0.000, C 0.000 }
gfCNCPoint1[22740] = {X 166.9493, Y 40.7947, Z -2.1667, A 0.000, B 0.000, C 0.000 }
gfCNCPoint1[22741] = {X 166.4848, Y 38.9932, Z -2.1667, A 0.000, B 0.000, C 0.000 }
gfCNCPoint1[22742] = {X 166.2300, Y 37.1503, Z -2.1667, A 0.000, B 0.000, C 0.000 }
gfCNCPoint1[22743] = {X 166.1316, Y 35.3979, Z -2.1667, A 0.000, B 0.000, C 0.000 }
gfCNCPoint1[22744] = {X 166.2083, Y 33.6444, Z -2.1667, A 0.000, B 0.000, C 0.000 }
gfCNCPoint1[22745] = {X 166.4593, Y 31.9074, Z -2.1667, A 0.000, B 0.000, C 0.000 }
gfCNCPoint1[22746] = {X 166.8821, Y 30.2039, Z -2.1667, A 0.000, B 0.000, C 0.000 }
gfCNCPoint1[22747] = {X 167.4726, Y 28.5511, Z -2.1667, A 0.000, B 0.000, C 0.000 }
gfCNCPoint1[22748] = {X 168.2335, Y 26.9819, Z -2.1667, A 0.000, B 0.000, C 0.000 }
gfCNCPoint1[22749] = {X 169.1859, Y 25.5210, Z -2.1667, A 0.000, B 0.000, C 0.000 }
gfCNCPoint1[22750] = {X 170.3147, Y 24.1916, Z -2.1667, A 0.000, B 0.000, C 0.000 }
gfCNCPoint1[22751] = {X 169.9867, Y 23.6226, Z -2.1667, A 0.000, B 0.000, C 0.000 }
gfCNCPoint1[22752] = {X 169.7112, Y 23.0263, Z -2.1667, A 0.000, B 0.000, C 0.000 }
gfCNCPoint1[22753] = {X 167.1001, Y 16.6309, Z -2.1667, A 0.000, B 0.000, C 0.000 }
gfCNCPoint1[22754] = {X 166.7820, Y 15.6636, Z -2.1667, A 0.000, B 0.000, C 0.000 }
gfCNCPoint1[22755] = {X 166.6021, Y 14.6613, Z -2.1667, A 0.000, B 0.000, C 0.000 }
gfCNCPoint1[22756] = {X 166.6021, Y 17.4615, Z -2.1667, A 0.000, B 0.000, C 0.000 }
gfCNCPoint1[22757] = {X 166.5130, Y 18.5970, Z -2.1667, A 0.000, B 0.000, C 0.000 }
gfCNCPoint1[22758] = {X 166.2479, Y 19.7047, Z -2.1667, A 0.000, B 0.000, C 0.000 }
gfCNCPoint1[22759] = {X 165.8132, Y 20.7575, Z -2.1667, A 0.000, B 0.000, C 0.000 }
gfCNCPoint1[22760] = {X 165.2197, Y 21.7296, Z -2.1667, A 0.000, B 0.000, C 0.000 }
gfCNCPoint1[22761] = {X 164.3788, Y 22.6988, Z -2.1667, A 0.000, B 0.000, C 0.000 }
gfCNCPoint1[22762] = {X 163.3807, Y 23.5052, Z -2.1667, A 0.000, B 0.000, C 0.000 }
gfCNCPoint1[22763] = {X 162.2566, Y 24.1239, Z -2.1667, A 0.000, B 0.000, C 0.000 }
gfCNCPoint1[22764] = {X 161.0414, Y 24.5356, Z -2.1667, A 0.000, B 0.000, C 0.000 }
gfCNCPoint1[22765] = {X 160.4746, Y 22.2035, Z -2.1667, A 0.000, B 0.000, C 0.000 }
gfCNCPoint1[22766] = {X 159.9024, Y 22.3069, Z -2.1667, A 0.000, B 0.000, C 0.000 }
gfCNCPoint1[22767] = {X 159.3220, Y 22.3415, Z -2.1667, A 0.000, B 0.000, C 0.000 }
gfCNCPoint1[22768] = {X 158.6806, Y 22.3415, Z -2.1667, A 0.000, B 0.000, C 0.000 }
gfCNCPoint1[22769] = {X 157.8824, Y 22.2731, Z -2.1667, A 0.000, B 0.000, C 0.000 }
gfCNCPoint1[22770] = {X 157.1059, Y 22.0760, Z -2.1667, A 0.000, B 0.000, C 0.000 }
gfCNCPoint1[22771] = {X 156.3717, Y 21.7554, Z -2.1667, A 0.000, B 0.000, C 0.000 }
gfCNCPoint1[22772] = {X 155.5229, Y 21.1776, Z -2.1667, A 0.000, B 0.000, C 0.000 }
gfCNCPoint1[22773] = {X 154.8127, Y 20.4361, Z -2.1667, A 0.000, B 0.000, C 0.000 }
gfCNCPoint1[22774] = {X 152.8357, Y 20.4371, Z -2.1667, A 0.000, B 0.000, C 0.000 }
gfCNCPoint1[22775] = {X 152.8341, Y 40.6542, Z -2.1667, A 0.000, B 0.000, C 0.000 }
gfCNCPoint1[22776] = {X 153.1756, Y 41.0235, Z -2.1667, A 0.000, B 0.000, C 0.000 }
gfCNCPoint1[22777] = {X 153.6801, Y 41.7282, Z -2.1667, A 0.000, B 0.000, C 0.000 }
gfCNCPoint1[22778] = {X 154.0531, Y 42.5104, Z -2.1667, A 0.000, B 0.000, C 0.000 }
gfCNCPoint1[22779] = {X 154.2832, Y 43.3459, Z -2.1667, A 0.000, B 0.000, C 0.000 }
gfCNCPoint1[22780] = {X 154.3631, Y 44.2089, Z -2.1667, A 0.000, B 0.000, C 0.000 }
gfCNCPoint1[22781] = {X 154.3629, Y 45.0469, Z -2.1667, A 0.000, B 0.000, C 0.000 }
gfCNCPoint1[22782] = {X 154.3440, Y 45.4308, Z -2.1667, A 0.000, B 0.000, C 0.000 }
gfCNCPoint1[22783] = {X 154.2951, Y 45.8119, Z -2.1667, A 0.000, B 0.000, C 0.000 }
gfCNCPoint1[22784] = {X 154.0370, Y 46.7541, Z -2.1667, A 0.000, B 0.000, C 0.000 }
gfCNCPoint1[22785] = {X 153.5963, Y 47.6260, Z -2.1667, A 0.000, B 0.000, C 0.000 }
gfCNCPoint1[22786] = {X 152.9909, Y 48.3926, Z -2.1667, A 0.000, B 0.000, C 0.000 }
gfCNCPoint1[22787] = {X 152.2448, Y 49.0233, Z -2.1667, A 0.000, B 0.000, C 0.000 }
gfCNCPoint1[22788] = {X 151.3881, Y 49.4928, Z -2.1667, A 0.000, B 0.000, C 0.000 }
gfCNCPoint1[22789] = {X 150.4551, Y 49.7822, Z -2.1667, A 0.000, B 0.000, C 0.000 }
gfCNCPoint1[22790] = {X 149.4831, Y 49.8800, Z -2.1667, A 0.000, B 0.000, C 0.000 }
gfCNCPoint1[22791] = {X 143.0396, Y 49.8800, Z -2.1667, A 0.000, B 0.000, C 0.000 }
gfCNCPoint1[22792] = {X 142.0923, Y 49.7872, Z -2.1667, A 0.000, B 0.000, C 0.000 }
gfCNCPoint1[22793] = {X 141.1811, Y 49.5122, Z -2.1667, A 0.000, B 0.000, C 0.000 }
gfCNCPoint1[22794] = {X 140.3405, Y 49.0656, Z -2.1667, A 0.000, B 0.000, C 0.000 }
gfCNCPoint1[22795] = {X 139.6026, Y 48.4643, Z -2.1667, A 0.000, B 0.000, C 0.000 }
gfCNCPoint1[22796] = {X 138.9955, Y 47.7312, Z -2.1667, A 0.000, B 0.000, C 0.000 }
gfCNCPoint1[22797] = {X 138.5423, Y 46.8942, Z -2.1667, A 0.000, B 0.000, C 0.000 }
gfCNCPoint1[22798] = {X 138.2601, Y 45.9852, Z -2.1667, A 0.000, B 0.000, C 0.000 }
gfCNCPoint1[22799] = {X 138.1598, Y 45.0386, Z -2.1667, A 0.000, B 0.000, C 0.000 }
gfCNCPoint1[22800] = {X 138.1601, Y 44.1416, Z -2.1667, A 0.000, B 0.000, C 0.000 }
gfCNCPoint1[22801] = {X 138.2148, Y 43.4769, Z -2.1667, A 0.000, B 0.000, C 0.000 }
gfCNCPoint1[22802] = {X 138.3597, Y 42.8258, Z -2.1667, A 0.000, B 0.000, C 0.000 }
gfCNCPoint1[22803] = {X 129.1532, Y 40.1052, Z -2.1667, A 0.000, B 0.000, C 0.000 }
gfCNCPoint1[22804] = {X 129.5665, Y 38.9035, Z -2.1667, A 0.000, B 0.000, C 0.000 }
gfCNCPoint1[22805] = {X 130.0836, Y 37.7426, Z -2.1667, A 0.000, B 0.000, C 0.000 }
gfCNCPoint1[22806] = {X 130.0836, Y 31.6021, Z -2.1667, A 0.000, B 0.000, C 0.000 }
gfCNCPoint1[22807] = {X 129.2058, Y 31.3796, Z -2.1667, A 0.000, B 0.000, C 0.000 }
gfCNCPoint1[22808] = {X 128.3436, Y 31.1026, Z -2.1667, A 0.000, B 0.000, C 0.000 }
gfCNCPoint1[22809] = {X 128.3433, Y 38.3276, Z -2.1667, A 0.000, B 0.000, C 0.000 }
gfCNCPoint1[22810] = {X 128.7842, Y 39.2000, Z -2.1667, A 0.000, B 0.000, C 0.000 }
